// TwinCAT 3 PLC project Theseus
// ProgramVersion: 3.1.4024.0
// libraries:
//   Tc2_ControllerToolbox, * (Beckhoff Automation GmbH)
//   Tc2_MC2, * (Beckhoff Automation GmbH)
//   Tc2_ModbusRTU, * (Beckhoff Automation GmbH)
//   Tc2_Standard, * (Beckhoff Automation GmbH)
//   Tc2_System, * (Beckhoff Automation GmbH)
//   Tc2_Utilities, * (Beckhoff Automation GmbH)
//   Tc3_Module, * (Beckhoff Automation GmbH)
//   Tc2_OpcUa,3.3.2.0,Beckhoff Automation GmbH
// project tree:
//   Data_Types/ E_MachineState.TcDUT, E_PIDMode.TcDUT (not stored), E_LMH.TcDUT, E_ProductType.TcDUT, E_Status.TcDUT
//   GVLs/ Global_Alarms.TcGVL, Global_Constants.TcGVL, P0_Global_Variables.TcGVL
//   / PlcTask.TcTTO (not stored)
//   POUs/ FB_Reactor.TcPOU, FB_Reactor_Set.TcPOU, MAIN.TcPOU, P_Alarms.TcPOU, P_M01.TcPOU, P_U01.TcPOU
//   POUs/Functions/ F_AnalogIn.TcPOU (not stored), F_Concat3.TcPOU (not stored), F_Concat4.TcPOU, F_HighestInt.TcPOU (not stored), F_IEConvert.TcPOU, F_LowestReal.TcPOU (not stored), F_HighestReal.TcPOU, F_LowMidHigh.TcPOU, F_Temperature.TcPOU (not stored), F_SetProcess.TcPOU (not stored), F_ValveClear.TcPOU
//   POUs/Function_Blocks/ FB_Analog_Out.TcPOU, FB_ChangeOfValue.TcPOU, FB_Door_Closed.TcPOU, FB_Integer_Out.TcPOU, FB_MovingAverage.TcPOU, FB_PI_Control.TcPOU, FB_RateOfChange.TcPOU, FB_Temperature.TcPOU, FB_ValveError.TcPOU, FB_VFD.TcPOU
// real-time tasks:
//   TASK PlcTask: cycle T#10ms, priority 20, ADS port 350
// I/O:
//   DEVICE Device 2 (EtherCAT) (disabled), AmsNetId 192.168.1.143.3.1
//     Term 1 (EK1100) [EK1100 EtherCAT Coupler (2A E-Bus)]
//       Term 2 (EL6070) [EL6070 1Ch. Licensing-Terminal]
//       Term 3 (EL1008) [EL1008 8Ch. Dig. Input 24V, 3ms]
//       Term 4 (EL1008) [EL1008 8Ch. Dig. Input 24V, 3ms]
//       Term 5 (EL1008) [EL1008 8Ch. Dig. Input 24V, 3ms]
//       Term 6 (EL1008) [EL1008 8Ch. Dig. Input 24V, 3ms]
//       Term 7 (EL1008) [EL1008 8Ch. Dig. Input 24V, 3ms]
//       Term 8 (EL1008) [EL1008 8Ch. Dig. Input 24V, 3ms]
//       Term 9 (EL1008) [EL1008 8Ch. Dig. Input 24V, 3ms]
//       Term 10 (EL2008) [EL2008 8Ch. Dig. Output 24V, 0.5A]
//       Term 11 (EL2008) [EL2008 8Ch. Dig. Output 24V, 0.5A]
//       Term 12 (EL2008) [EL2008 8Ch. Dig. Output 24V, 0.5A]
//       Term 13 (EL2008) [EL2008 8Ch. Dig. Output 24V, 0.5A]
//       Term 14 (EL2008) [EL2008 8Ch. Dig. Output 24V, 0.5A]
//       Term 15 (EL2008) [EL2008 8Ch. Dig. Output 24V, 0.5A]
//       Term 16 (EL2008) [EL2008 8Ch. Dig. Output 24V, 0.5A]
//       Term 18 (EL9410) [EL9410 E-Bus Power Supplier  (Diagnostics)]
//       Term 19 (EL3058) [EL3058 8Ch. Ana. Input 4-20mA]
//       Term 20 (EL3058) [EL3058 8Ch. Ana. Input 4-20mA]
//       Term 21 (EL3058) [EL3058 8Ch. Ana. Input 4-20mA]
//       Term 22 (EL3058) [EL3058 8Ch. Ana. Input 4-20mA]
//       Term 23 (EL3058) [EL3058 8Ch. Ana. Input 4-20mA]
//       Term 24 (EL4122) [EL4122 2Ch. Ana. Output  4-20mA, 16bit]
//       Term 25 (EL3318) [EL3318 8Ch. Ana Input Thermocouple (TC)]
//       Term 26 (EL3318) [EL3318 8Ch. Ana Input Thermocouple (TC)]
//       Term 27 (EL3318) [EL3318 8Ch. Ana Input Thermocouple (TC)]
//       Term 28 (EL3318) [EL3318 8Ch. Ana Input Thermocouple (TC)]
//       Term 29 (EL3318) [EL3318 8Ch. Ana Input Thermocouple (TC)]
//       Term 30 (EL9410) [EL9410 E-Bus Power Supplier  (Diagnostics)]
//       Term 31 (EL3214) [EL3214 4Ch. Ana. Input PT100 (RTD)]
//       Term 32 (EK1110) [EK1110 EtherCAT extension]
//     Term 33 (EK1100) [EK1100 EtherCAT Coupler (2A E-Bus)]
//       Term 34 (EL3058) [EL3058 8Ch. Ana. Input 4-20mA]
//       Term 35 (EL3058) [EL3058 8Ch. Ana. Input 4-20mA]
//       Term 36 (EL2008) [EL2008 8Ch. Dig. Output 24V, 0.5A]
//       Term 37 (EL2008) [EL2008 8Ch. Dig. Output 24V, 0.5A]
//       Term 38 (EK1122) [EK1122 2 port EtherCAT junction]
//         Box 40 (Commander C200 Open Loop) [Commander C200 Open Loop]
//       Term 39 (EL9011) [EL9011 End Terminal]
// variable links:
//   Theseus/Theseus Instance <-> Device 2 (EtherCAT)/Term 1 (EK1100)/Term 10 (EL2008)
//     PlcTask Outputs/P_M01.rs1.r1.AT_01_pump <-> Channel 3/Output
//     PlcTask Outputs/P_M01.rs1.r1.AT_03_pump <-> Channel 1/Output
//     PlcTask Outputs/P_M01.rs1.r1.AT_01_sol <-> Channel 4/Output
//     PlcTask Outputs/P_M01.rs1.r1.AT_03_sol <-> Channel 2/Output
//     PlcTask Outputs/P_M01.rs1.r1.XV_02 <-> Channel 5/Output
//     PlcTask Outputs/P_M01.rs1.r1.XV_09 <-> Channel 6/Output
//     PlcTask Outputs/P_M01.rs1.r1.outlet_door_far_clamps_extend_valve <-> Channel 7/Output
//     PlcTask Outputs/P_M01.rs1.r1.outlet_door_far_clamps_retract_valve <-> Channel 8/Output
//   Theseus/Theseus Instance <-> Device 2 (EtherCAT)/Term 1 (EK1100)/Term 11 (EL2008)
//     PlcTask Outputs/P_M01.rs1.r1.inlet_door_far_clamps_extend_valve <-> Channel 3/Output
//     PlcTask Outputs/P_M01.rs1.r1.inlet_door_far_clamps_retract_valve <-> Channel 4/Output
//     PlcTask Outputs/P_M01.rs1.r1.inlet_door_near_clamps_extend_valve <-> Channel 5/Output
//     PlcTask Outputs/P_M01.rs1.r1.inlet_door_near_clamps_retract_valve <-> Channel 6/Output
//     PlcTask Outputs/P_M01.rs1.r1.outlet_door_close_valve <-> Channel 8/Output
//     PlcTask Outputs/P_M01.rs1.r1.outlet_door_near_clamps_extend_valve <-> Channel 1/Output
//     PlcTask Outputs/P_M01.rs1.r1.outlet_door_near_clamps_retract_valve <-> Channel 2/Output
//     PlcTask Outputs/P_M01.rs1.r1.outlet_door_open_valve <-> Channel 7/Output
//   Theseus/Theseus Instance <-> Device 2 (EtherCAT)/Term 1 (EK1100)/Term 12 (EL2008)
//     PlcTask Outputs/P_M01.rs1.XV_04 <-> Channel 3/Output
//     PlcTask Outputs/P_M01.rs1.XV_05 <-> Channel 4/Output
//     PlcTask Outputs/P_M01.rs1.XV_06 <-> Channel 5/Output
//     PlcTask Outputs/P_M01.rs1.XV_07 <-> Channel 6/Output
//     PlcTask Outputs/P_M01.rs1.XV_08 <-> Channel 7/Output
//     PlcTask Outputs/P_M01.rs1.r1.inlet_door_close_valve <-> Channel 2/Output
//     PlcTask Outputs/P_M01.rs1.r1.inlet_door_open_valve <-> Channel 1/Output
//   Theseus/Theseus Instance <-> Device 2 (EtherCAT)/Term 1 (EK1100)/Term 13 (EL2008)
//     PlcTask Outputs/P_U01.XV_03 <-> Channel 4/Output
//     PlcTask Outputs/P_U01.XV_04 <-> Channel 3/Output
//     PlcTask Outputs/P_U01.XV_06 <-> Channel 1/Output
//     PlcTask Outputs/P_U01.XV_12 <-> Channel 6/Output
//   Theseus/Theseus Instance <-> Device 2 (EtherCAT)/Term 1 (EK1100)/Term 14 (EL2008)
//     PlcTask Outputs/P_U01.XV_10 <-> Channel 1/Output
//     PlcTask Outputs/P_U01.XV_11 <-> Channel 4/Output
//     PlcTask Outputs/P_U01.XV_13 <-> Channel 2/Output
//     PlcTask Outputs/P_U01.XV_14 <-> Channel 5/Output
//   Theseus/Theseus Instance <-> Device 2 (EtherCAT)/Term 1 (EK1100)/Term 19 (EL3058)
//     PlcTask Inputs/P_M01.rs1.r1.AT_01 <-> AI Standard Channel 3/Value
//     PlcTask Inputs/P_M01.rs1.r1.AT_02 <-> AI Standard Channel 2/Value
//     PlcTask Inputs/P_M01.rs1.r1.AT_03 <-> AI Standard Channel 1/Value
//     PlcTask Inputs/P_M01.rs1.r1.AT_04 <-> AI Standard Channel 4/Value
//     PlcTask Inputs/P_M01.rs1.r1.AT_01_error <-> AI Standard Channel 1/Status/Error
//     PlcTask Inputs/P_M01.rs1.r1.AT_02_error <-> AI Standard Channel 2/Status/Error
//     PlcTask Inputs/P_M01.rs1.r1.AT_03_error <-> AI Standard Channel 3/Status/Error
//     PlcTask Inputs/P_M01.rs1.r1.AT_04_error <-> AI Standard Channel 4/Status/Error
//     PlcTask Inputs/P_M01.rs1.r1.FT_01 <-> AI Standard Channel 5/Value
//     PlcTask Inputs/P_M01.rs1.r1.FT_01_error <-> AI Standard Channel 5/Status/Error
//     PlcTask Inputs/P_M01.rs1.r1.PDT_01 <-> AI Standard Channel 6/Value
//     PlcTask Inputs/P_M01.rs1.r1.PDT_02 <-> AI Standard Channel 7/Value
//     PlcTask Inputs/P_M01.rs1.r1.PDT_03 <-> AI Standard Channel 8/Value
//     PlcTask Inputs/P_M01.rs1.r1.PDT_01_error <-> AI Standard Channel 6/Status/Error
//     PlcTask Inputs/P_M01.rs1.r1.PDT_02_error <-> AI Standard Channel 7/Status/Error
//     PlcTask Inputs/P_M01.rs1.r1.PDT_03_error <-> AI Standard Channel 8/Status/Error
//   Theseus/Theseus Instance <-> Device 2 (EtherCAT)/Term 1 (EK1100)/Term 20 (EL3058)
//     PlcTask Inputs/P_M01.rs1.FT_02 <-> AI Standard Channel 2/Value
//     PlcTask Inputs/P_M01.rs1.FT_02_error <-> AI Standard Channel 2/Status/Error
//     PlcTask Inputs/P_M01.rs1.PT_02 <-> AI Standard Channel 3/Value
//     PlcTask Inputs/P_M01.rs1.PT_02_error <-> AI Standard Channel 3/Status/Error
//     PlcTask Inputs/P_M01.rs1.r1.PT_01 <-> AI Standard Channel 1/Value
//     PlcTask Inputs/P_M01.rs1.r1.PT_01_error <-> AI Standard Channel 1/Status/Error
//     PlcTask Inputs/P_U01.WI_01 <-> AI Standard Channel 4/Value
//     PlcTask Inputs/P_U01.WI_02 <-> AI Standard Channel 5/Value
//     PlcTask Inputs/P_U01.WI_03 <-> AI Standard Channel 6/Value
//     PlcTask Inputs/P_U01.WI_01_error <-> AI Standard Channel 4/Status/Error
//     PlcTask Inputs/P_U01.WI_02_error <-> AI Standard Channel 5/Status/Error
//     PlcTask Inputs/P_U01.WI_03_error <-> AI Standard Channel 6/Status/Error
//   Theseus/Theseus Instance <-> Device 2 (EtherCAT)/Term 1 (EK1100)/Term 21 (EL3058)
//     PlcTask Inputs/P_U01.AT_02 <-> AI Standard Channel 6/Value
//     PlcTask Inputs/P_U01.AT_03 <-> AI Standard Channel 7/Value
//     PlcTask Inputs/P_U01.AT_02_error <-> AI Standard Channel 6/Status/Error
//     PlcTask Inputs/P_U01.AT_03_error <-> AI Standard Channel 7/Status/Error
//     PlcTask Inputs/P_U01.FT_02 <-> AI Standard Channel 8/Value
//     PlcTask Inputs/P_U01.FT_04 <-> AI Standard Channel 1/Value
//     PlcTask Inputs/P_U01.FT_07 <-> AI Standard Channel 5/Value
//     PlcTask Inputs/P_U01.FT_02_error <-> AI Standard Channel 8/Status/Error
//     PlcTask Inputs/P_U01.FT_04_error <-> AI Standard Channel 1/Status/Error
//     PlcTask Inputs/P_U01.FT_07_error <-> AI Standard Channel 5/Status/Error
//     PlcTask Inputs/P_U01.LT_02 <-> AI Standard Channel 4/Value
//     PlcTask Inputs/P_U01.LT_02_error <-> AI Standard Channel 4/Status/Error
//     PlcTask Inputs/P_U01.PCV_01_position <-> AI Standard Channel 3/Value
//     PlcTask Inputs/P_U01.PT_04 <-> AI Standard Channel 2/Value
//     PlcTask Inputs/P_U01.PT_04_error <-> AI Standard Channel 2/Status/Error
//     PlcTask Inputs/P_U01.vacuum_pres_control_valve_position_error <-> AI Standard Channel 3/Status/Error
//   Theseus/Theseus Instance <-> Device 2 (EtherCAT)/Term 1 (EK1100)/Term 22 (EL3058)
//     PlcTask Inputs/P_U01.FT_05 <-> AI Standard Channel 1/Value
//     PlcTask Inputs/P_U01.FT_06 <-> AI Standard Channel 4/Value
//     PlcTask Inputs/P_U01.FT_08 <-> AI Standard Channel 7/Value
//     PlcTask Inputs/P_U01.FT_05_error <-> AI Standard Channel 1/Status/Error
//     PlcTask Inputs/P_U01.FT_06_error <-> AI Standard Channel 4/Status/Error
//     PlcTask Inputs/P_U01.FT_08_error <-> AI Standard Channel 7/Status/Error
//     PlcTask Inputs/P_U01.LT_01 <-> AI Standard Channel 2/Value
//     PlcTask Inputs/P_U01.LT_01_error <-> AI Standard Channel 2/Status/Error
//     PlcTask Inputs/P_U01.PCV_02_position <-> AI Standard Channel 3/Value
//     PlcTask Inputs/P_U01.PDT_04 <-> AI Standard Channel 6/Value
//     PlcTask Inputs/P_U01.PDT_04_error <-> AI Standard Channel 6/Status/Error
//     PlcTask Inputs/P_U01.PT_07 <-> AI Standard Channel 5/Value
//     PlcTask Inputs/P_U01.PT_07_error <-> AI Standard Channel 5/Status/Error
//   Theseus/Theseus Instance <-> Device 2 (EtherCAT)/Term 1 (EK1100)/Term 24 (EL4122)
//     PlcTask Outputs/P_U01.PCV_01 <-> Channel 1/Output
//     PlcTask Outputs/P_U01.PCV_02 <-> Channel 2/Output
//   Theseus/Theseus Instance <-> Device 2 (EtherCAT)/Term 1 (EK1100)/Term 25 (EL3318)
//     PlcTask Inputs/P_M01.rs1.r1._01_TT_01 <-> TC Channel 1/Value
//     PlcTask Inputs/P_M01.rs1.r1._01_TT_03 <-> TC Channel 2/Value
//     PlcTask Inputs/P_M01.rs1.r1._02_TT_01 <-> TC Channel 3/Value
//     PlcTask Inputs/P_M01.rs1.r1._02_TT_03 <-> TC Channel 4/Value
//     PlcTask Inputs/P_M01.rs1.r1._03_TT_01 <-> TC Channel 5/Value
//     PlcTask Inputs/P_M01.rs1.r1._03_TT_03 <-> TC Channel 6/Value
//     PlcTask Inputs/P_M01.rs1.r1._04_TT_01 <-> TC Channel 7/Value
//     PlcTask Inputs/P_M01.rs1.r1._04_TT_03 <-> TC Channel 8/Value
//     PlcTask Inputs/P_M01.rs1.r1._01_TT_01_Error <-> TC Channel 1/Status/Error
//     PlcTask Inputs/P_M01.rs1.r1._01_TT_03_Error <-> TC Channel 2/Status/Error
//     PlcTask Inputs/P_M01.rs1.r1._02_TT_01_Error <-> TC Channel 3/Status/Error
//     PlcTask Inputs/P_M01.rs1.r1._02_TT_03_Error <-> TC Channel 4/Status/Error
//     PlcTask Inputs/P_M01.rs1.r1._03_TT_01_Error <-> TC Channel 5/Status/Error
//     PlcTask Inputs/P_M01.rs1.r1._03_TT_03_Error <-> TC Channel 6/Status/Error
//     PlcTask Inputs/P_M01.rs1.r1._04_TT_01_Error <-> TC Channel 7/Status/Error
//     PlcTask Inputs/P_M01.rs1.r1._04_TT_03_Error <-> TC Channel 8/Status/Error
//   Theseus/Theseus Instance <-> Device 2 (EtherCAT)/Term 1 (EK1100)/Term 26 (EL3318)
//     PlcTask Inputs/P_M01.rs1.r1._05_TT_01 <-> TC Channel 1/Value
//     PlcTask Inputs/P_M01.rs1.r1._05_TT_03 <-> TC Channel 2/Value
//     PlcTask Inputs/P_M01.rs1.r1._06_TT_01 <-> TC Channel 3/Value
//     PlcTask Inputs/P_M01.rs1.r1._06_TT_03 <-> TC Channel 4/Value
//     PlcTask Inputs/P_M01.rs1.r1._07_TT_01 <-> TC Channel 5/Value
//     PlcTask Inputs/P_M01.rs1.r1._07_TT_03 <-> TC Channel 6/Value
//     PlcTask Inputs/P_M01.rs1.r1._08_TT_01 <-> TC Channel 7/Value
//     PlcTask Inputs/P_M01.rs1.r1._08_TT_03 <-> TC Channel 8/Value
//     PlcTask Inputs/P_M01.rs1.r1._05_TT_01_Error <-> TC Channel 1/Status/Error
//     PlcTask Inputs/P_M01.rs1.r1._05_TT_03_Error <-> TC Channel 2/Status/Error
//     PlcTask Inputs/P_M01.rs1.r1._06_TT_01_Error <-> TC Channel 3/Status/Error
//     PlcTask Inputs/P_M01.rs1.r1._06_TT_03_Error <-> TC Channel 4/Status/Error
//     PlcTask Inputs/P_M01.rs1.r1._07_TT_01_Error <-> TC Channel 5/Status/Error
//     PlcTask Inputs/P_M01.rs1.r1._07_TT_03_Error <-> TC Channel 6/Status/Error
//     PlcTask Inputs/P_M01.rs1.r1._08_TT_01_Error <-> TC Channel 7/Status/Error
//     PlcTask Inputs/P_M01.rs1.r1._08_TT_03_Error <-> TC Channel 8/Status/Error
//   Theseus/Theseus Instance <-> Device 2 (EtherCAT)/Term 1 (EK1100)/Term 27 (EL3318)
//     PlcTask Inputs/P_M01.rs1.r1._09_TT_01 <-> TC Channel 1/Value
//     PlcTask Inputs/P_M01.rs1.r1._09_TT_03 <-> TC Channel 2/Value
//     PlcTask Inputs/P_M01.rs1.r1._10_TT_01 <-> TC Channel 3/Value
//     PlcTask Inputs/P_M01.rs1.r1._10_TT_03 <-> TC Channel 4/Value
//     PlcTask Inputs/P_M01.rs1.r1._11_TT_01 <-> TC Channel 5/Value
//     PlcTask Inputs/P_M01.rs1.r1._11_TT_03 <-> TC Channel 6/Value
//     PlcTask Inputs/P_M01.rs1.r1._12_TT_01 <-> TC Channel 7/Value
//     PlcTask Inputs/P_M01.rs1.r1._12_TT_03 <-> TC Channel 8/Value
//     PlcTask Inputs/P_M01.rs1.r1._09_TT_01_Error <-> TC Channel 1/Status/Error
//     PlcTask Inputs/P_M01.rs1.r1._09_TT_03_Error <-> TC Channel 2/Status/Error
//     PlcTask Inputs/P_M01.rs1.r1._10_TT_01_Error <-> TC Channel 3/Status/Error
//     PlcTask Inputs/P_M01.rs1.r1._10_TT_03_Error <-> TC Channel 4/Status/Error
//     PlcTask Inputs/P_M01.rs1.r1._11_TT_01_Error <-> TC Channel 5/Status/Error
//     PlcTask Inputs/P_M01.rs1.r1._11_TT_03_Error <-> TC Channel 6/Status/Error
//     PlcTask Inputs/P_M01.rs1.r1._12_TT_01_Error <-> TC Channel 7/Status/Error
//     PlcTask Inputs/P_M01.rs1.r1._12_TT_03_Error <-> TC Channel 8/Status/Error
//   Theseus/Theseus Instance <-> Device 2 (EtherCAT)/Term 1 (EK1100)/Term 29 (EL3318)
//     PlcTask Inputs/P_M01.rs1.TT_01 <-> TC Channel 1/Value
//     PlcTask Inputs/P_M01.rs1.TT_01_error <-> TC Channel 1/Status/Error
//     PlcTask Inputs/P_U01.TT_03 <-> TC Channel 2/Value
//     PlcTask Inputs/P_U01.TT_06 <-> TC Channel 5/Value
//     PlcTask Inputs/P_U01.TT_10 <-> TC Channel 3/Value
//     PlcTask Inputs/P_U01.TT_11 <-> TC Channel 4/Value
//     PlcTask Inputs/P_U01.TT_03_error <-> TC Channel 2/Status/Error
//     PlcTask Inputs/P_U01.TT_06_error <-> TC Channel 5/Status/Error
//     PlcTask Inputs/P_U01.TT_10_error <-> TC Channel 3/Status/Error
//     PlcTask Inputs/P_U01.TT_11_error <-> TC Channel 4/Status/Error
//   Theseus/Theseus Instance <-> Device 2 (EtherCAT)/Term 1 (EK1100)/Term 3 (EL1008)
//     PlcTask Inputs/P_M01.rs1.r1.outlet_door_far_clamps_extended <-> Channel 6/Input
//     PlcTask Inputs/P_M01.rs1.r1.outlet_door_far_closed_ls <-> Channel 4/Input
//     PlcTask Inputs/P_M01.rs1.r1.outlet_door_far_open_ls <-> Channel 3/Input
//     PlcTask Inputs/P_M01.rs1.r1.outlet_door_near_clamps_extended <-> Channel 5/Input
//     PlcTask Inputs/P_M01.rs1.r1.outlet_door_near_closed_ls <-> Channel 2/Input
//     PlcTask Inputs/P_M01.rs1.r1.outlet_door_near_open_ls <-> Channel 1/Input
//     PlcTask Inputs/P_M01.rs1.r1.repres_valve_closed <-> Channel 8/Input
//     PlcTask Inputs/P_M01.rs1.r1.repres_valve_open <-> Channel 7/Input
//   Theseus/Theseus Instance <-> Device 2 (EtherCAT)/Term 1 (EK1100)/Term 31 (EL3214)
//     PlcTask Inputs/P_M01.rs1.r1.TT_04 <-> RTD Inputs Channel 2/Value
//     PlcTask Inputs/P_M01.rs1.r1.TT_05 <-> RTD Inputs Channel 1/Value
//     PlcTask Inputs/P_M01.rs1.r1.TT_04_error <-> RTD Inputs Channel 2/Status/Error
//     PlcTask Inputs/P_M01.rs1.r1.TT_05_error <-> RTD Inputs Channel 1/Status/Error
//     PlcTask Inputs/P_U01.TT_02 <-> RTD Inputs Channel 3/Value
//     PlcTask Inputs/P_U01.TT_02_error <-> RTD Inputs Channel 3/Status/Error
//   Theseus/Theseus Instance <-> Device 2 (EtherCAT)/Term 1 (EK1100)/Term 4 (EL1008)
//     PlcTask Inputs/P_M01.rs1.r1.inlet_door_far_clamps_extended <-> Channel 6/Input
//     PlcTask Inputs/P_M01.rs1.r1.inlet_door_far_closed_ls <-> Channel 4/Input
//     PlcTask Inputs/P_M01.rs1.r1.inlet_door_far_open_ls <-> Channel 3/Input
//     PlcTask Inputs/P_M01.rs1.r1.inlet_door_near_clamps_extended <-> Channel 5/Input
//     PlcTask Inputs/P_M01.rs1.r1.inlet_door_near_closed_ls <-> Channel 2/Input
//     PlcTask Inputs/P_M01.rs1.r1.inlet_door_near_open_ls <-> Channel 1/Input
//     PlcTask Inputs/P_M01.rs1.reactor_drain_vessel_lsh <-> Channel 8/Input
//     PlcTask Inputs/P_M01.rs1.reactor_drain_vessel_lsl <-> Channel 7/Input
//   Theseus/Theseus Instance <-> Device 2 (EtherCAT)/Term 1 (EK1100)/Term 5 (EL1008)
//     PlcTask Inputs/P_M01.rs1.condensate_valve_closed <-> Channel 6/Input
//     PlcTask Inputs/P_M01.rs1.condensate_valve_open <-> Channel 5/Input
//     PlcTask Inputs/P_M01.rs1.dead_air_valve_closed <-> Channel 2/Input
//     PlcTask Inputs/P_M01.rs1.dead_air_valve_open <-> Channel 1/Input
//     PlcTask Inputs/P_M01.rs1.product_iso_valve_closed <-> Channel 4/Input
//     PlcTask Inputs/P_M01.rs1.product_iso_valve_open <-> Channel 3/Input
//     PlcTask Inputs/P_M01.rs1.steam_iso_valve_closed <-> Channel 8/Input
//     PlcTask Inputs/P_M01.rs1.steam_iso_valve_open <-> Channel 7/Input
//   Theseus/Theseus Instance <-> Device 2 (EtherCAT)/Term 1 (EK1100)/Term 6 (EL1008)
//     PlcTask Inputs/P_M01.rs1.steam_bypass_valve_closed <-> Channel 2/Input
//     PlcTask Inputs/P_M01.rs1.steam_bypass_valve_open <-> Channel 1/Input
//   Theseus/Theseus Instance <-> Device 2 (EtherCAT)/Term 1 (EK1100)/Term 7 (EL1008)
//     PlcTask Inputs/P_U01.knockout_drain_valve_closed <-> Channel 4/Input
//     PlcTask Inputs/P_U01.knockout_drain_valve_open <-> Channel 3/Input
//     PlcTask Inputs/P_U01.product_condensate_drum_lsh <-> Channel 2/Input
//     PlcTask Inputs/P_U01.product_condensate_drum_lsl <-> Channel 1/Input
//     PlcTask Inputs/P_U01.vacuum_pump_bypass_valve_closed <-> Channel 6/Input
//     PlcTask Inputs/P_U01.vacuum_pump_bypass_valve_open <-> Channel 5/Input
//     PlcTask Inputs/P_U01.vacuum_pump_inlet_valve_closed <-> Channel 8/Input
//     PlcTask Inputs/P_U01.vacuum_pump_inlet_valve_open <-> Channel 7/Input
//   Theseus/Theseus Instance <-> Device 2 (EtherCAT)/Term 1 (EK1100)/Term 8 (EL1008)
//     PlcTask Inputs/P_U01.dead_air_inlet_valve_closed <-> Channel 2/Input
//     PlcTask Inputs/P_U01.dead_air_inlet_valve_open <-> Channel 1/Input
//     PlcTask Inputs/P_U01.product_line_ambient_valve_ambient <-> Channel 5/Input
//     PlcTask Inputs/P_U01.product_line_ambient_valve_product <-> Channel 6/Input
//     PlcTask Inputs/P_U01.separator_drain_valve_closed <-> Channel 4/Input
//     PlcTask Inputs/P_U01.separator_drain_valve_open <-> Channel 3/Input
//   Theseus/Theseus Instance <-> Device 2 (EtherCAT)/Term 33 (EK1100)/Term 34 (EL3058)
//     PlcTask Inputs/P_U01.IT1 <-> AI Standard Channel 5/Value
//     PlcTask Inputs/P_U01.IT2 <-> AI Standard Channel 6/Value
//     PlcTask Inputs/P_U01.IT3 <-> AI Standard Channel 7/Value
//     PlcTask Inputs/P_U01.IT4 <-> AI Standard Channel 8/Value
//     PlcTask Inputs/P_U01.VT1 <-> AI Standard Channel 1/Value
//     PlcTask Inputs/P_U01.VT2 <-> AI Standard Channel 2/Value
//     PlcTask Inputs/P_U01.VT3 <-> AI Standard Channel 3/Value
//     PlcTask Inputs/P_U01.VT4 <-> AI Standard Channel 4/Value
//     PlcTask Inputs/P_U01.l1_current_120_error <-> AI Standard Channel 8/Status/Error
//     PlcTask Inputs/P_U01.l1_current_240_error <-> AI Standard Channel 5/Status/Error
//     PlcTask Inputs/P_U01.l2_current_240_error <-> AI Standard Channel 6/Status/Error
//     PlcTask Inputs/P_U01.l3_current_240_error <-> AI Standard Channel 7/Status/Error
//     PlcTask Inputs/P_U01.l1_voltage_120_error <-> AI Standard Channel 4/Status/Error
//     PlcTask Inputs/P_U01.l1_voltage_240_error <-> AI Standard Channel 1/Status/Error
//     PlcTask Inputs/P_U01.l2_voltage_240_error <-> AI Standard Channel 2/Status/Error
//     PlcTask Inputs/P_U01.l3_voltage_240_error <-> AI Standard Channel 3/Status/Error
//   Theseus/Theseus Instance <-> Device 2 (EtherCAT)/Term 33 (EK1100)/Term 36 (EL2008)
//     PlcTask Outputs/P_U01.B_01 <-> Channel 5/Output
//     PlcTask Outputs/P_U01.P_01 <-> Channel 4/Output
//     PlcTask Outputs/P_U01.P_02 <-> Channel 2/Output
//     PlcTask Outputs/P_U01.P_03 <-> Channel 1/Output
//     PlcTask Outputs/P_U01.P_05 <-> Channel 7/Output
//     PlcTask Outputs/P_U01.P_06 <-> Channel 3/Output
//     PlcTask Outputs/P_U01.X_01 <-> Channel 8/Output
//     PlcTask Outputs/P_U01.boiler_reset <-> Channel 6/Output
//   Theseus/Theseus Instance <-> Device 2 (EtherCAT)/Term 33 (EK1100)/Term 37 (EL2008)
//     PlcTask Outputs/P_U01.E_01 <-> Channel 2/Output
//     PlcTask Outputs/P_U01.P_04 <-> Channel 1/Output
//   Theseus/Theseus Instance <-> Device 2 (EtherCAT)/Term 33 (EK1100)/Term 38 (EK1122)/Box 40 (Commander C200 Open Loop)
//     PlcTask Inputs/P_M01.rs1.r1.fan_vfd_current <-> Transmit PDO Mapping 6/vfd output current param 04_001
//     PlcTask Inputs/P_M01.rs1.r1.fan_vfd_ecat_state <-> WcState/WcState
//     PlcTask Inputs/P_M01.rs1.r1.fan_vfd_status <-> Transmit PDO Mapping 6/Status word
//     PlcTask Inputs/P_M01.rs1.r1.fan_vfd_velocity <-> Transmit PDO Mapping 6/vl velocity actual value
//     PlcTask Outputs/P_M01.rs1.r1.fan_vfd_control <-> Receive PDO Mapping 6/Control word
//     PlcTask Outputs/P_M01.rs1.r1.fan_vfd_target_vel <-> Receive PDO Mapping 6/vl target velocity

// ---- Data_Types/E_MachineState.TcDUT
// Theseus - E_MachineState
// Rev 1.0 - December 2, 2024

TYPE E_MachineState :
(
	eStateOff						:= 0,
	eIdle,
	eDoorCycle,
	ePositivePressure,
	eRepressurization,
	eAdsorption,
	eEvacuation,
	eDesorption,
	eBypass,
	eSingleProcessAuto,
	eChangeState,
	ePause
);
END_TYPE

// ---- Data_Types/E_LMH.TcDUT
// Theseus - E_LMH
// Rev 1.0 - March 14, 2024

TYPE E_LMH :
(
	eLow			 													:= 0,
	eMid,
	eHigh
);
END_TYPE

// ---- Data_Types/E_ProductType.TcDUT
// Theseus - E_ProductType
// Rev 1.0 - June 15, 2024

TYPE E_ProductType :
(
	eAmbient			 												:= 0,
	eProduct
);
END_TYPE

// ---- Data_Types/E_Status.TcDUT
// Theseus - E_Status
// Rev 1.0 - December 2, 2024

TYPE E_Status :
(
	eSystem_Idle						:= 0,
	e1,
	e2,
	eWarmup_Running,			
	eSteamBypass_Running,		
	eDoorCycle_Running,		
	ePositivePressure_Running,	
	eRepressurization_Running,	
	eAdsorption_Running,		
	eEvacuation_Running,		
	eDesorption_Running,
	eBypass_Running,
	eShutting_Down,				
	ePressureTest_Running,		
	e12,                        
	eWarmup_Error,				
	eSteamBypass_Error,			
	eDoor_Cycle_Error,			
	ePositivePressure_Error,	
	eRepressurization_Error,	
	eAdsorption_Error,			
	eEvacuation_Error,			
	eDesorption_Error,
	eShutdown_Error,			
	ePressureTest_Error,		
	e21,                        
	e22,                        
	eWarmup_Complete,			
	eSteamBypass_Complete,		
	eDoorCycle_Complete,         
	ePositivePressure_Complete,	
	eRepressurization_Complete,	
	eAdsorption_Complete,		
	eEvacuation_Complete,		
	eDesorption_Complete,
	eBypass_Complete,		
	eShutdown_Complete,			
	ePressureTest_Complete,		
	e32,                        
	eStopping_Process,			
	eResetting,					
	eSaving_Data				
);
END_TYPE

// ---- GVLs/Global_Alarms.TcGVL
// Theseus - Global_Alarms
// Rev 1.0 - December 3, 2024

VAR_GLOBAL
	
	giAlarmCount														: INT		:= 0;
	gsAlarms															: ARRAY[0.._ALARM_COUNT] OF STRING;
	gsMessages															: ARRAY[0.._ALARM_COUNT] OF STRING;

	gsClampsNotExtendedError											: STRING	:= 'Clamps not extended';
	gsClampsNotRetractedError											: STRING	:= 'Clamps not retracted';
	gsDoorsNotSelectedError												: STRING	:= 'No doors were selected';
	gsGasketNotActivatedError											: STRING	:= 'Gasket not activated';
	gsInletDoorNotClosedError											: STRING	:= 'Inlet door not closed';
	gsInletDoorNotOpenError												: STRING	:= 'Inlet door not open';
	gsOutletDoorNotClosedError											: STRING	:= 'Outlet door not closed';
	gsOutletDoorNotOpenError											: STRING	:= 'Outlet door not open';
	gsPositivePressureError												: STRING	:= 'Reactor failed to reach positive pressure set point';
	gsReactorNotAtAmbientPressure										: STRING	:= 'Reactor not at ambient pressure';
	gsUnacceptableReactorLeakRate										: STRING	:= 'Unacceptable reactor positive pressure leak rate';
	gsRepressurizationValveError										: STRING	:= 'Repressurization valve error (XV02)';	

	
	gsAmbientPressureError												: STRING	:= 'Ambient pressure error';
	gsAdsorptionAcceptableButNotIdealTimeError							: STRING	:= 'Adsorption time to cool acceptable but not ideal';
	gsAdsorptionTimeOutError											: STRING	:= 'Adsorption - sorbent failed to cool';
	gsAdsorptionUnacceptableTimeError									: STRING	:= 'Adsorption time to cool unacceptable';
	gsAdsorptionInletCo2LowError										: STRING	:= 'Adsorption inlet co2 concentration low';
	gsAirFlowSensorError												: STRING	:= 'Air flow sensor error (R1 FT01)';
	gsBoilerError														: STRING	:= 'Boiler error';
	gsInletLineTempSensorError											: STRING	:= 'Inlet line temperature sensor error (TT06)';
	gsClampExtendError													: STRING	:= 'Clamp extend error';
	gsClampRetractError													: STRING	:= 'Clamp retract error';
	gsCondensateFlowSensorError											: STRING	:= 'Condensate flow sensor error (FT-04)';
	gsCondenserKODrainageError											: STRING	:= 'Condensate knockout drainage error';
	gsCondensateLslError												: STRING	:= 'Condensate low limit switch error (LS-01)';
	gsCondenserFlowSensorError											: STRING	:= 'Condenser flow sensor error (FT08)';
	gsCondensateProductDrainError										: STRING	:= 'Module product/cooling line not draining';	
	gsCondensateValveError												: STRING	:= 'Condensate valve error (XV06)';
	gsDeadAirInletValveError											: STRING	:= 'Dead air inlet valve error (XV10)';
	gsDeadAirLinePressureError											: STRING	:= 'Dead air line failed to reach desired pressure';
	gsDeadAirValveError													: STRING	:= 'Dead air valve error (XV04)';
	gsDesiredCycleCountError											: STRING	:= 'Desired cycle count error';
	gsDesorptionHighSteamLineTemp										: STRING	:= 'Desorption - High steam line temperature';
	gsDesorptionPurgeLinePressureError									: STRING	:= 'Desorption - Unable to purge';
	gsDoorClampsExtendedError											: STRING	:= 'Door clamps extended';
	gsDoorsNotClosedError												: STRING	:= 'Door not closed error';
	gsDoorsNotOpenError													: STRING	:= 'Door not open error';
	gsFanDiffPresSensorError											: STRING	:= 'Fan differential pressure sensor error (PDT-03)';
	gsFilterDiffPresSensorError											: STRING	:= 'Filter differential pressure sensor error (PDT-01)';
	gsFlowCalibrationDiffPresSensorError								: STRING	:= 'Flow calibration differential pressure sensor error (PDT04)';
	gsHighTempCountError												: STRING	:= 'High Temp Count Error';
	gsInletAirHighTempCountError										: STRING	:= 'Inlet air high temperature count error';
    gsInletCO2SensorError												: STRING	:= 'Inlet CO2 sensor error (AT-01)';
    gsInletH2OSensorError												: STRING	:= 'Inlet H2O sensor error (AT-02)';
	gsInletDoorClampsExtendedError										: STRING	:= 'Inlet door clamps extended error (XV01)'; 
	gsInletDoorClampsRetractedError										: STRING	:= 'Inlet door clamps retracted error (XV01)'; 
	gsNoReactorSetsSelected												: STRING	:= 'No reactor sets selected';
    gsOutletCO2SensorError												: STRING	:= 'Outlet CO2 sensor error (AT-03)';
    gsOutletH2OSensorError												: STRING	:= 'Outlet H2O sensor error (AT-04)';
	gsOutletDoorClampsExtendedError										: STRING	:= 'Outlet door clamps extended error (XV03)'; 
	gsOutletDoorClampsRetractedError									: STRING	:= 'Outlet door clamps retracted error (XV03)'; 
	gsProductVacuumTempSensorError										: STRING	:= 'Product vacuum temperature sensor error (TT-03)';
	gsProductTempSensorError											: STRING	:= 'Product temperature sensor error (TT-02)';
	gsProductCondensateDrainError										: STRING	:= 'Product condensate not draining';
	gsProductCondensateDrainValveError									: STRING	:= 'Product condensate drain valve error';
	gsProductCondensateDrumLshError										: STRING	:= 'Product condensate drum high limit switch error (LS-02)';
	gsProductCondensateDrumLslError										: STRING	:= 'Product condensate drum low limit switch error (LS-01)';
	gsProductLineAmbientValveError										: STRING	:= 'Product line ambient valve error (XV11)';
	gsProductLinePressureSensorError									: STRING	:= 'Product line pressure sensor error (PT02)';
	gsProductLineTempTooLowError										: string	:= 'Product line temperature too low';
	gsProductOutletH2oSensorError										: STRING	:= 'Product outlet h2o sensor error (AT-02B)';
	gsProductOutletCo2SensorError										: STRING	:= 'Product outlet co2 sensor error (AT-02A)';
	gsProductOutletFlowSensorError										: STRING	:= 'Product outlet flow sensor error (FT02)';
	gsProductVacuumBackfeedValveError									: STRING	:= 'Product vacuum backfeed valve error (PCV-01)';
	gsProductVacuumOutletIsoValveError									: STRING	:= 'Product vacuum outlet isolation valve error (XV-05)';
	gsProductVacuumPumpIsoValveError									: STRING	:= 'Product vacuum pump isolation valve error (XV-03)';
	gsProductVacuumPresSensorError										: STRING	:= 'Product vacuum pressure sensor error (PT-05)';
	gsPurgeProductLinePresLowError										: STRING	:= 'Purge product line pressure low error';
	gsProductIsoValveError												: STRING	:= 'Product isolation valve error (XV05)';
	gsProductLinePresSensorError										: STRING	:= 'Product line pressure sensor error (PT-02)';
	gsProductLineTempSensorError										: STRING	:= 'Product line temperature sensor error (TT-01)';
	gsReactorCondensateFlowSensorError									: STRING	:= 'Reactor condensate flow sensor error (FT02)';
	gsReactorDrainError													: STRING	:= 'Reactor not draining';	
	gsReactorDoorClosingError											: STRING	:= 'Failed to close door valves';									// Complete
	gsReactorDoorOpeningError											: STRING	:= 'Failed to open door valves';									// Complete
	gsReactorsAtAmbientPressure											: STRING	:= 'Reactors at ambient pressure';
	gsReactorPressureAboveAcceptableLevelError							: STRING	:= 'Reactor pressure above acceptable level';
	gsReactorPressureAboveDesiredLevelError								: STRING	:= 'Reactor pressure above desired level';
	gsReactorPressureTooHighError										: STRING	:= 'Reactor pressure too high error';
	gsReactorPressureTooLowError										: STRING	:= 'Reactor pressure too low error';
	gsReactorPresSensorError											: STRING	:= 'Reactor pressure sensor error (PT01)';
	gsReactorSetFailedToPressurizeError									: STRING	:= 'Reactor set failed to pressurize';
	gsReactorValvesNotClosedError										: STRING	:= 'Reactor valves are not closed';
	gsRepressurizationError												: STRING	:= 'Repressurization error';	
	gsSorbentDiffPresSensorError										: STRING	:= 'Sorbent differential pressure sensor error (PDT-02)';
	gsSorbentTemperatureError											: STRING	:= 'Sorbent temperatures above safe temperature';
	gsSteamBypassMinFlowRateError										: STRING	:= 'Steam bypass minimum flow rate error';
	gsSteamControlValveError											: STRING	:= 'Steam control valve error (PCV-01)';
	gsSteamIsoValveError												: STRING	:= 'Steam isolation valve error (XV07)';
	gsSteamFailedToPressurizeReactorError								: STRING	:= 'Steam failed to pressurize reactor to purge pressure';
	gsSteamFlowSensorError												: STRING	:= 'Steam flow sensor error (FT05)';
	gsSteamBypassValveError												: STRING	:= 'Steam bypass valve error (XV08)';
	gsSteamPressureHighError											: STRING	:= 'High steam pressure';
	gsSteamPressureLowError												: STRING	:= 'Low steam pressure';
	gsSteamTemperatureLowError											: STRING	:= 'Low steam temperature';
	gsSteamLinePresSensorError											: STRING	:= 'Steam line pressure sensor error (PT07)';
	gsSteamFlowConrolValveError											: STRING	:= 'Steam flow control valve error (PCV02)';
	gsSteamFlowTooLowError												: STRING	:= 'Steam flow too low error';
	gsSteamWaterTankLevelSensorError									: STRING	:= 'Steam water tank level sensor error (LT01)';
	gsTapWaterFeedFlowSensorError										: STRING	:= 'Tap water feed flow sensor error (FT05)';
	gsUnableToEvacuateLinesError										: STRING	:= 'Unable to evacuate lines in time';
	gsVacuumPressureControlValveError									: STRING	:= 'Vacuum pressure control valve error (PCV01)';
	gsVacuumCoolingLoopFlowError										: STRING	:= 'Vacuum cooling loop flow error';
	gsVacuumCoolingLoopTempError										: STRING	:= 'Vacuum cooling loop temperature error';
	gsVacuumCoolingUnacceptableError									: STRING	:= 'Vacuum cooling temperature reached was unacceptable';
	gsVacuumCoolingAcceptableButNotIdealError							: STRING	:= 'Vacuum cooling temperature reached was acceptable but not ideal';
	gsVacuumLinePressureHighError										: STRING	:= 'Vacuum line pressure high';
	gsVacuumPumpWaterFlowSensorError									: STRING	:= 'Vacuum pump water flow sensor error (FT07)';
	gsVacuumPumpWaterTemp1SensorError									: STRING	:= 'Vacuum pump water temperature 1 sensor error (TT10)';
	gsVacuumPressureUnacceptableError									: STRING	:= 'Vacuum pressure reached was unacceptable';
	gsVacuumPressureAcceptableBotNotIdealError							: STRING	:= 'Vacuum pressure reached was acceptable but not ideal';
	gsVacuumPumpBypassValveError										: STRING	:= 'Vacuum pump bypass valve error (XV04)';
	gsVacuumPumpInletValveError											: STRING	:= 'Vacuum pump inlet valve error (XV03)';
	gsVacuumSeparatorLevelSensorError									: STRING	:= 'Vacuum separator level sensor error (LT02)';
	gsVacuumSeparatorDrainError											: STRING	:= 'Vacuum separator drain error';
	gsVacuumSeparatorFillError											: STRING	:= 'Vacuum separator fill error';
	gsWarmupNotRunError													: STRING	:= 'Warmup has not run';
	gsWeatherHumiditySensorError										: STRING	:= 'Weather humidity sensor error (AT-07)';
	gsWeatherPresureSensorError											: STRING	:= 'Weather pressure sensor error (PT-09)';
	gsWaterScale1SensorError											: STRING	:= 'Water Scale 1 sensor error (WI-01)';
	gsWaterScale2SensorError											: STRING	:= 'Water Scale 2 sensor error (WI-02)';
	gsWaterScale3SensorError											: STRING	:= 'Water Scale 3 sensor error (WI-03)';
	
	gsMessageTBD			: STRING	:= 'TBD';
	gsAdsorptionCo2LowCheck												: STRING	:= 'Check inlet co2 sensor';
	gsCheckOperation													: STRING	:= 'Check sensor operation';
	gsExtraRepressurizationTimeAllowed									: STRING	:= 'Extra repressurization time allowed';
	gsPressureDropTestCannotRun											: STRING	:= 'Pressure drop test cannot run';
	gsProcessCannotContinue												: STRING	:= 'Process cannot continue';
	gsProcessCannotRun													: STRING	:= 'Process cannot run';
	gsProcessCannotRunAdsorptionWillContinue							: STRING	:= 'Process cannot run - Adsorption will continue';
	gsProcessStopsAtEOA													: STRING	:= 'Process will stop at end of Adsorption';
	gsProcessStopsAtEOC													: STRING	:= 'Process will stop at end of current cycle';
	gsProcessWillContinue												: STRING	:= 'Process will continue';
	gsProcessComplete													: STRING	:= 'Process complete';
	gsProcessRestart													: STRING	:= 'Process will attempt to restart on next cycle';
	gsReactorIsUnderVacuum												: STRING	:= 'Reactor is under vacuum';
	gsReactorSetCannotRun												: STRING	:= 'Reactor set cannot run';
	gsReactorSetWillContinue											: STRING	:= 'Reactor set will continue';
	gsReactorSetWillPause												: STRING	:= 'Reactor set will pause';
	gsReactorSetWillStop												: STRING	:= 'Reactor set will stop';
	gsReactorSetWillStopAtEndOfCycle									: STRING	:= 'Reactor set will stop at end of cycle';
	gsReactorSetsInEvacuationWillContinue								: STRING	:= 'Reactor sets in Evacuation will finish, others will stop';
	gsReactorSetWillStopEvacWillFinishOthersWillCompleteCycle			: STRING	:= 'Reactor set will stop, Evacuation will finish, others will complete cycle';
	gsRunWarmup															: STRING	:= 'Run warm up';													
	gsSorbentDamaged													: STRING	:= 'Sorbent damaged';
	gsSteamBypassWillContinueWOAdsorption								: STRING	:= 'Steam Bypass will continue without Adsorption';
	gsSystemCannotRun													: STRING	:= 'System cannot run';
	gsSystemWillStop													: STRING	:= 'System will stop';
	gsSystemWillStopAfterDesorption										: STRING	:= 'System will stop after Desorption';
	gsUnableToCloseDoors												: STRING	:= 'Unable to close doors';
	gsUnableToEvacuateReactorSet										: STRING	:= 'Unable to evacuate reactor set';
	gsUserProcessRestart												: STRING	:= 'User must restart for process to continue';
	gsWarmupWillContinue												: STRING	:= 'Warm up will continue';													
	gsWarmupWillContinueWOAdsorption									: STRING	:= 'Warm up will continue without Adsorption';
	gsWarning															: STRING	:= 'Waring - Procees could be affected';

END_VAR

// ---- GVLs/Global_Constants.TcGVL
// Theseus - Global_Constants
// Rev 1.0 - November 4, 2024

VAR_GLOBAL CONSTANT
	
	_DOOR_ACTUATION_TIMEOUT												: REAL		:= 120000;
	_CLAMP_ACTUATION_TIMEOUT											: REAL		:= 10000;
	_VALVE_TIME															: REAL		:= 5000;
	
	_ALARM_COUNT														: INT		:= 100;
	_DRAIN_TIME															: TIME		:= T#3S;
	_DOOR_LATCH_CLOSE_TIME												: TIME		:= T#2S;
	_FAN_SPEED_MAX														: REAL		:= 1765;		// Maximum Fan RPM
	_FAN_SPEED_MIN														: REAL		:= 300;			// Minimum Fan RPM
	_PUMP_SPEED_MAX														: REAL		:= 3540;		// Maximum Pump RPM
	_PUMP_SPEED_MIN														: REAL		:= 200;			// Minimum Pump RPM
	_FAN_DELAY_TIME														: INT		:= 2000;
	_FAN_RS_DELAY_TIME													: INT		:= 15000;
	_PROCESS_COMPLETE_TIME												: REAL		:= 2000;
	_PAUSE_TIME															: REAL		:= 2000;
	_FAN_SHUTDOWN_TIME													: REAL		:= 10000;
	_VALVE_INCREMENT_TIME												: REAL		:= 250;			// Time period for incremental change in valve position (mSecs)
	_STOPPING_TIME														: REAL		:= 2000;
	_VALVE_CLOSED														: INT		:= 3;
	_VALVE_OPEN															: INT		:= 95;
	
	_CURRENT_120_FACTOR													: REAL		:= 655.34;		// =  32767 counts / 50 amps
	_CURRENT_240_FACTOR													: REAL		:= 218.44;      // = 32767 counts / 150 amps
	_CURRENT_BOILER_FACTOR												: REAL 		:= 40.95 * 2 ;	//  = 32767 / 800 Amps * 2 (double coiled)
	_CURRENT_MODULE_FACTOR												: REAL		:= 81.91;		// 0- 800 amps	
	_PERCENT_FACTOR														: REAL		:= 327.67;		// Factor to convert input to output percentage
	_FAN_RPM_FACTOR														: REAL		:= 17.65;		// Factor to convert fan percent input to rpm output (max rpm / 100)
	_PUMP_RPM_FACTOR													: REAL		:= 35.4;		// Factor to convert pump percent input to rpm output (max rpm / 100)
	_BLOWER_RPM_FACTOR													: REAL      := 34.7;		// product blower rpm = 3470
	_VOLTAGE_120_FACTOR													: REAL		:= 218.44;		// 0- 150 VAC
	_VOLTAGE_240_FACTOR													: REAL		:= 65.53;		// 0 - 500 VAC 
	
	_INLET_AIR_MAX_COUNT												: INT		:= 0;
	_ADSORP_MAX_COUNT													: INT		:= 1;
	_VAC_COOLING_MAX_COUNT												: INT		:= 1;
	_DESORP_MAX_COUNT													: INT		:= 1;
	_HIGH_CART_READINGS_MAX												: INT		:= 2;
	_RETRY_ATTEMPTS														: INT		:= 3;
	_MAX_REACTOR_ERRORS													: INT		:= 3;
	
	_PRESSURE_PERCENT													: REAL		:= 0.9;
	_TEMP_DEADBAND														: REAL		:= 0.5;
	
	_TIMEOUT_WARMUP_RESET												: TIME		:= T#10M;
	_TIMEOUT_RESET														: TIME		:= T#3S;
	
	_OPEN																: INT 		:= 100;
	_CLOSED																: INT		:= 0;

	_SECONDS															: REAL		:= 1000;
	_MINUTES															: REAL		:= 60000;
	
	_U01																: STRING	:= 'U01 - ';
	_RS01																: STRING	:= 'RS01 - ';
	_R1																	: STRING	:= 'Reactor1';
	
	STEAM_TABLE  : ARRAY[1..30] OF ARRAY [0..1] OF REAL := [[0.0,0.0],[0.02,0.000015],[0.03,0.000022],[0.04,0.000029],[0.05,0.000035],[0.06,0.000042],[0.07,0.000049],[0.08,0.000055],[0.09,0.000062],
															[0.1,0.000068],[0.2,0.000131],[0.3,0.000191],[0.4,0.00025],[0.5,0.000309],[0.6,0.000366],[0.7,0.000423],[0.8,0.000479],[0.9,0.000535],
															[1.0,0.00059],[1.1,0.000645],[1.2,0.0007],[1.3,0.000755],[1.4,0.000809],[1.5,0.000863],[1.6,0.000916],[1.7,0.00097],[1.8,0.001023],[1.8,0.001023],[1.9,0.001076],
															[2.0,0.001129]];

END_VAR

// ---- GVLs/P0_Global_Variables.TcGVL
// Theseus - Global_Variables
// Rev 1.0 - October 2, 2024

VAR_GLOBAL

	gbRS01TestError														: BOOL;
	gbRS02TestError														: BOOL;
	gbRS03TestError														: BOOL;
	
	gbDrainageOn														: BOOL;
	gbCondenserKODrainageOn												: BOOL;
	gbCondensateValve													: BOOL;
	
	gbGasketsActivated													: BOOL;
	gbFirstEvacuation													: BOOL;
	giEvacuationCounter													: INT;

	gsCycleMode															: STRING;
	gsCycleStage														: STRING;
	gsM01RS01CycleStage													: STRING;
	gsM01RS02CycleStage													: STRING;
	gsM01RS03CycleStage													: STRING;
	
	gbRepresValves														: BOOL;
	
END_VAR

// ---- POUs/FB_Reactor.TcPOU
FUNCTION_BLOCK FB_Reactor
VAR_INPUT
	
	unit																: INT;

    /// <summary>XV01</summary>
	{attribute 'OPC.UA.DA' := '1'}  				                
	open_inlet_door														: BOOL;
    /// <summary>XV01</summary>
	{attribute 'OPC.UA.DA' := '1'}  				                
	close_inlet_door													: BOOL;
    /// <summary>XV03</summary>
	{attribute 'OPC.UA.DA' := '1'}  				                
	open_outlet_door													: BOOL;
    /// <summary>XV03</summary>
	{attribute 'OPC.UA.DA' := '1'}  				                
	close_outlet_door													: BOOL;

    /// <summary>XV01</summary>
	{attribute 'OPC.UA.DA' := '1'}  				                
	extend_inlet_door_clamps											: BOOL;
    /// <summary>XV01</summary>
	{attribute 'OPC.UA.DA' := '1'}  				                
	retract_inlet_door_clamps											: BOOL;
    /// <summary>XV03</summary>
	{attribute 'OPC.UA.DA' := '1'}  				                
	extend_outlet_door_clamps											: BOOL;
    /// <summary>XV03</summary>
	{attribute 'OPC.UA.DA' := '1'}  				                
	retract_outlet_door_clamps											: BOOL;

	/// <summary>XV02</summary>
	{attribute 'OPC.UA.DA' := '1'}  				                
	repres_valve														: BOOL;
	/// <summary>XV09</summary>
	{attribute 'OPC.UA.DA' := '1'}  				                
	over_pressure_test_control											: BOOL;
	
	/// <summary>AT01_pump</summary>
	{attribute 'OPC.UA.DA' := '1'}  				                
	inlet_co2_pump														: BOOL;
    /// <summary>AT01_solenoid</summary>
	{attribute 'OPC.UA.DA' := '1'}  				                
	inlet_co2_sol														: BOOL;

    /// <summary>AT03_pump</summary>
	{attribute 'OPC.UA.DA' := '1'}  				                
	outlet_co2_pump														: BOOL;
    /// <summary>AT03_solenoid</summary>
	{attribute 'OPC.UA.DA' := '1'}  				                
	outlet_co2_sol														: BOOL;
	
    /// <summary>F01</summary>
	fan_vfd_setpoint													: REAL;

END_VAR
VAR_OUTPUT

	inlet_doors_open													: BOOL;
    outlet_doors_open													: BOOL;	
    inlet_doors_closed													: BOOL;	
    outlet_doors_closed													: BOOL;	

	inlet_door_clamps_extended											: BOOL;
	inlet_door_clamps_retracted											: BOOL;
	outlet_door_clamps_extended											: BOOL;
    outlet_door_clamps_retracted										: BOOL;
	
	sorbent_low_temp													: REAL;
	sorbent_high_temp													: REAL;
	sorbent_average_temp												: REAL;

	desorption_high_temp_count											: INT;
	adsorption_high_temp_count											: INT;
	vacuum_cooling_high_temp_count										: INT;

    /// <summary>AT01</summary>																			// Summary defines hover over text while in twincat 3 program
	{attribute 'OPC.UA.DA' := '1'}  				                									// OPC_UA tag
	{attribute 'OPC.UA.DA.Access' := '1'}																// OPC_UA tag definition - '1' indicates Read Only, '2' indicates Write Only (not used), '3' indicates Read Write (default)  				                
	inlet_co2															: REAL;							// Tag value to read (scaled)
    /// <summary>AT01</summary>
	{attribute 'OPC.UA.DA' := '1'}  				                
	{attribute 'OPC.UA.DA.Access' := '1'}  				                
	inlet_co2_error														: BOOL;

    /// <summary>AT02</summary>
	{attribute 'OPC.UA.DA' := '1'}  				                
	{attribute 'OPC.UA.DA.Access' := '1'}  				                
	inlet_h2o															: REAL;
    /// <summary>AT02</summary>
	{attribute 'OPC.UA.DA' := '1'}  				                
	{attribute 'OPC.UA.DA.Access' := '1'}  				                
	inlet_h2o_error														: BOOL;

    /// <summary>AT03</summary>
	{attribute 'OPC.UA.DA' := '1'}
	{attribute 'OPC.UA.DA.Access' := '1'}  				                
	outlet_co2															: REAL;
    /// <summary>AT03</summary>
	{attribute 'OPC.UA.DA' := '1'}  				                
	{attribute 'OPC.UA.DA.Access' := '1'}  				                
	outlet_co2_error													: BOOL;

    /// <summary>AT04</summary>
	{attribute 'OPC.UA.DA' := '1'}  				                
	{attribute 'OPC.UA.DA.Access' := '1'}  				                
	outlet_h2o															: REAL;
    /// <summary>AT04</summary>
	{attribute 'OPC.UA.DA' := '1'}  				                
	{attribute 'OPC.UA.DA.Access' := '1'}  				                
	outlet_h2o_error													: BOOL;

    /// <summary>PT01</summary>
	{attribute 'OPC.UA.DA' := '1'}  				                
	{attribute 'OPC.UA.DA.Access' := '1'}  				                
	reactor_pres														: REAL;
    /// <summary>PT01</summary>
	{attribute 'OPC.UA.DA' := '1'}  				                
	{attribute 'OPC.UA.DA.Access' := '1'}  				                
	reactor_pres_error													: BOOL;

    /// <summary>FT01</summary>
	{attribute 'OPC.UA.DA' := '1'}  				                
	{attribute 'OPC.UA.DA.Access' := '1'}  				                
	air_flow															: REAL;
    /// <summary>FT01</summary>
	{attribute 'OPC.UA.DA' := '1'}  				                
	{attribute 'OPC.UA.DA.Access' := '1'}  				                
	air_flow_error														: BOOL;

    /// <summary>PDT01</summary>
	{attribute 'OPC.UA.DA' := '1'}  				                
	{attribute 'OPC.UA.DA.Access' := '1'}  				                
	filter_diff_pres													: REAL;
    /// <summary>PDT01</summary>
	{attribute 'OPC.UA.DA' := '1'}  				                
	{attribute 'OPC.UA.DA.Access' := '1'}  				                
	filter_diff_pres_error												: BOOL;

    /// <summary>PDT02</summary>
	{attribute 'OPC.UA.DA' := '1'}  				                
	{attribute 'OPC.UA.DA.Access' := '1'}  				                
	sorbent_diff_pres													: REAL;
    /// <summary>PDT02</summary>
	{attribute 'OPC.UA.DA' := '1'}  				                
	{attribute 'OPC.UA.DA.Access' := '1'}  				                
	sorbent_diff_pres_error												: BOOL;

    /// <summary>PDT03</summary>
	{attribute 'OPC.UA.DA' := '1'}  				                
	{attribute 'OPC.UA.DA.Access' := '1'}  				                
	fan_diff_pres														: REAL;
    /// <summary>PDT03</summary>
	{attribute 'OPC.UA.DA' := '1'}  				                
	{attribute 'OPC.UA.DA.Access' := '1'}  				                
	fan_diff_pres_error													: BOOL;
    /// <summary>TT04</summary>
	{attribute 'OPC.UA.DA' := '1'}  				                
	{attribute 'OPC.UA.DA.Access' := '1'}  				                
	air_inlet_temp														: REAL;
    /// <summary>TT04</summary>
	{attribute 'OPC.UA.DA' := '1'}  				                
	{attribute 'OPC.UA.DA.Access' := '1'}  				                
	air_inlet_temp_error												: BOOL;
	
    /// <summary>TT05</summary>
	{attribute 'OPC.UA.DA' := '1'}  				                
	{attribute 'OPC.UA.DA.Access' := '1'}  				                
	reactor_wall_temp													: REAL;
    /// <summary>Reactor Wall Temp</summary>
	{attribute 'OPC.UA.DA' := '1'}  				                
	{attribute 'OPC.UA.DA.Access' := '1'}  				                
	reactor_wall_temp_error												: BOOL;
	
    /// <summary>AT01_pump</summary>
	{attribute 'OPC.UA.DA' := '1'}  				                
	{attribute 'OPC.UA.DA.Access' := '1'}  				                
	inlet_co2_pump_cmd_status											: BOOL;
    /// <summary>AT01_solenoid</summary>
	{attribute 'OPC.UA.DA' := '1'}  				                
	{attribute 'OPC.UA.DA.Access' := '1'}  				                
	inlet_co2_sol_cmd_status											: BOOL;

    /// <summary>AT03_pump</summary>
	{attribute 'OPC.UA.DA' := '1'}  				                
	{attribute 'OPC.UA.DA.Access' := '1'}  				                
	outlet_co2_pump_cmd_status											: BOOL;
    /// <summary>AT03_solenoid</summary>
	{attribute 'OPC.UA.DA' := '1'}  				                
	{attribute 'OPC.UA.DA.Access' := '1'}  				                
	outlet_co2_sol_cmd_status											: BOOL;
	
    /// <summary>XV-02</summary>
	repres_valve_clear													: BOOL;

    /// <summary>XV09</summary>
	{attribute 'OPC.UA.DA' := '1'}  				                
	{attribute 'OPC.UA.DA.Access' := '1'}  				                
	over_pressure_test_control_cmd_status								: BOOL;

END_VAR
VAR
	fb_Fan																: FB_VFD();
	tonFan																: TON;
	rRpm																: REAL;
	rFanSPOld															: REAL			:= 0;

	fbInletDoorsClosed													: FB_Door_Closed();
	fbOutletDoorsClosed													: FB_Door_Closed();
	
	rtrigSorbentErrorCheck												: R_TRIG;
	i																	: INT;
	iCount																: ARRAY [0..23] OF INT;

	iInletAirSetpoint													: INT			:= 0;
	iTempCount															: INT;
	iHighTempCount														: INT;
	rTempTotal															: REAL;
	rTempSP																: REAL;
	rMin																: REAL;
	rMax																: REAL;

	cart01_temp_front_calc												: FB_Temperature;
	cart01_temp_back_calc												: FB_Temperature;
	cart02_temp_front_calc												: FB_Temperature;
	cart02_temp_back_calc												: FB_Temperature;
	cart03_temp_front_calc												: FB_Temperature;
	cart03_temp_back_calc												: FB_Temperature;
	cart04_temp_front_calc												: FB_Temperature;
	cart04_temp_back_calc												: FB_Temperature;
	cart05_temp_front_calc												: FB_Temperature;
	cart05_temp_back_calc												: FB_Temperature;
	cart06_temp_front_calc												: FB_Temperature;
	cart06_temp_back_calc												: FB_Temperature;
	cart07_temp_front_calc												: FB_Temperature;
	cart07_temp_back_calc												: FB_Temperature;
	cart08_temp_front_calc												: FB_Temperature;
	cart08_temp_back_calc												: FB_Temperature;
	cart09_temp_front_calc												: FB_Temperature;
	cart09_temp_back_calc												: FB_Temperature;
	cart10_temp_front_calc												: FB_Temperature;
	cart10_temp_back_calc												: FB_Temperature;
	cart11_temp_front_calc												: FB_Temperature;
	cart11_temp_back_calc												: FB_Temperature;
	cart12_temp_front_calc												: FB_Temperature;
	cart12_temp_back_calc												: FB_Temperature;
	
    /// <summary>AT01</summary>
	{attribute 'OPC.UA.DA' := '1'}  				                
	_InletCO2ErrorOff													: BOOL;
    /// <summary>Inlet CO2</summary>
	AT_01														AT %I*	: INT;
    /// <summary>Inlet CO2</summary>
	{attribute 'OPC.UA.DA' := '1'}
	{attribute 'OPC.UA.DA.Access' := '1'}  				                
	AT_01_error													AT %I*	: BOOL;

    /// <summary>AT02</summary>
	{attribute 'OPC.UA.DA' := '1'}  				                
	_InletH2OErrorOff													: BOOL;
    /// <summary>Inlet H20</summary>
	AT_02														AT %I*	: INT;
    /// <summary>Inlet H20</summary>
	{attribute 'OPC.UA.DA' := '1'}  				                
	{attribute 'OPC.UA.DA.Access' := '1'}  				                
	AT_02_error													AT %I*	: BOOL;

    /// <summary>AT03</summary>
	{attribute 'OPC.UA.DA' := '1'}  				                
	_OutletCO2ErrorOff													: BOOL;
    /// <summary>Outlet CO2</summary>
	AT_03														AT %I*	: INT;
    /// <summary>Outlet CO2</summary>
	{attribute 'OPC.UA.DA' := '1'}
	{attribute 'OPC.UA.DA.Access' := '1'}  				                
	AT_03_error													AT %I*	: BOOL;

    /// <summary>AT04</summary>
	{attribute 'OPC.UA.DA' := '1'}  				                
	_OutletH2OErrorOff													: BOOL;
    /// <summary>Outlet H20</summary>
	AT_04														AT %I*	: INT;
    /// <summary>Outlet H20</summary>
	{attribute 'OPC.UA.DA' := '1'}  				                
	{attribute 'OPC.UA.DA.Access' := '1'}  				                
	AT_04_error													AT %I*	: BOOL;

    /// <summary>PT01</summary>
	{attribute 'OPC.UA.DA' := '1'}
	_ReactorPresErrorOff												: BOOL;  				                
    /// <summary>Reactor Pressure</summary>
	PT_01														AT %I*	: INT;
    /// <summary>Reactor Pressure</summary>
	{attribute 'OPC.UA.DA' := '1'}  				                
	{attribute 'OPC.UA.DA.Access' := '1'}  				                
	PT_01_error													AT %I*	: BOOL;

    /// <summary>FT01</summary>
	{attribute 'OPC.UA.DA' := '1'}  				                
	_AirFlowErrorOff													: BOOL;
    /// <summary>Air flow</summary>
	FT_01														AT %I*	: INT;
    /// <summary>Air flow</summary>
	{attribute 'OPC.UA.DA' := '1'}  				                
	{attribute 'OPC.UA.DA.Access' := '1'}  				                
	FT_01_error													AT %I*	: BOOL;

    /// <summary>PDT01</summary>
	{attribute 'OPC.UA.DA' := '1'}  				                
	_FilterDiffPresErrorOff												: BOOL;
    /// <summary>Filter diff pres</summary>
	PDT_01														AT %I*	: INT;
    /// <summary>Filter diff pres</summary>
	{attribute 'OPC.UA.DA' := '1'}  				                
	{attribute 'OPC.UA.DA.Access' := '1'}  				                
	PDT_01_error												AT %I*	: BOOL;

    /// <summary>PDT02</summary>
	{attribute 'OPC.UA.DA' := '1'}  				                
	_SorbentDiffPresErrorOff											: BOOL;
    /// <summary>Sorbent diff pres</summary>
	PDT_02														AT %I*	: INT;
    /// <summary>Sorbent diff pres</summary>
	{attribute 'OPC.UA.DA' := '1'}  				                
	{attribute 'OPC.UA.DA.Access' := '1'}  				                
	PDT_02_error												AT %I*	: BOOL;

    /// <summary>PDT03</summary>
	{attribute 'OPC.UA.DA' := '1'}  				                
	_FanDiffPresErrorOff												: BOOL;
    /// <summary>fan diff pres</summary>
	PDT_03														AT %I*	: INT;
    /// <summary>fan diff pres</summary>
	{attribute 'OPC.UA.DA' := '1'}  				                
	{attribute 'OPC.UA.DA.Access' := '1'}  				                
	PDT_03_error												AT %I*	: BOOL;
	
    /// <summary>TT04</summary>
	{attribute 'OPC.UA.DA' := '1'}  				                
	_AirInletTempErrorOff												: BOOL;
    /// <summary>air inlet temp</summary>
	TT_04														AT %I*	: INT;
    /// <summary>air inlet temp</summary>
	{attribute 'OPC.UA.DA' := '1'}  				                
	{attribute 'OPC.UA.DA.Access' := '1'}  				                
	TT_04_error													AT %I*	: BOOL;

    /// <summary>TT05</summary>
	_ReactorWallTempErrorOff											: BOOL;
    /// <summary>Reactor wall temp</summary>
	TT_05														AT %I*	: INT;
    /// <summary>Reactor wall temp</summary>
	{attribute 'OPC.UA.DA' := '1'}  				                
	{attribute 'OPC.UA.DA.Access' := '1'}  				                
	TT_05_error													AT %I*	: BOOL;
	
    /// <summary>Inlet CO2 pump</summary>
	AT_01_pump													AT %Q*	: BOOL;
    /// <summary>Inlet CO2 solenoid</summary>
	AT_01_sol													AT %Q*	: BOOL;

    /// <summary>Inlet CO2 pump</summary>
	AT_03_pump													AT %Q*	: BOOL;
    /// <summary>Outlet CO2 solenoid</summary>
	AT_03_sol													AT %Q*	: BOOL;

    /// <summary>XV02</summary>
	{attribute 'OPC.UA.DA' := '1'}  				                
	{attribute 'OPC.UA.DA.Access' := '1'}  				                
	repres_valve_open_cmd_status										: BOOL;
    /// <summary>XV02</summary>
	{attribute 'OPC.UA.DA' := '1'}  				                
	{attribute 'OPC.UA.DA.Access' := '1'}  				                
	repres_valve_open											AT %I*	: BOOL;
    /// <summary>XV02</summary>
	{attribute 'OPC.UA.DA' := '1'}  				                
	{attribute 'OPC.UA.DA.Access' := '1'}  				                
	repres_valve_closed											AT %I*	: BOOL;
    /// <summary>repres valve</summary>
	XV_02														AT %Q*	: BOOL;
	
    /// <summary>over pressure test control</summary>
	XV_09														AT %Q*	: BOOL;
	
    /// <summary>F01</summary>
	{attribute 'OPC.UA.DA' := '1'}  				                
	fan_vfd_enable														: BOOL :=  TRUE;
    /// <summary>F01</summary>
	{attribute 'OPC.UA.DA' := '1'}  				                
	fan_vfd_reset														: BOOL;
    /// <summary>F01</summary>
	{attribute 'OPC.UA.DA' := '1'}  				                
	{attribute 'OPC.UA.DA.Access' := '1'}  				                
	fan_vfd_enabled														: BOOL;
    /// <summary>F01</summary>
	{attribute 'OPC.UA.DA' := '1'}  				                
	{attribute 'OPC.UA.DA.Access' := '1'}  				                
	fan_vfd_error														: BOOL;
    /// <summary>F01</summary>
	{attribute 'OPC.UA.DA' := '1'}  				                
	{attribute 'OPC.UA.DA.Access' := '1'}  				                
	fan_vfd_output														: REAL;
	 /// <summary>F01</summary>
	{attribute 'OPC.UA.DA' := '1'}  				                
	{attribute 'OPC.UA.DA.Access' := '1'}  				                
	fan_vfd_output_current												: REAL;
    /// <summary>F01</summary>
	fan_vfd_control												AT %Q*	: WORD;
    /// <summary>F01</summary>
	fan_vfd_target_vel											AT %Q*	: WORD;
    /// <summary>F01</summary>
	fan_vfd_status												AT %I*	: WORD;
    /// <summary>F01</summary>
	fan_vfd_velocity											AT %I*	: WORD;
    /// <summary>F01</summary>
	fan_vfd_ecat_state											AT %I*  : BOOL;
	fan_vfd_current												AT %I*	: DINT;
	//fan_vfd_current_amps										AT %Q*	: REAL;

    /// <summary>XV01_SV05</summary>
	inlet_door_open_valve										AT %Q*	: BOOL;
    /// <summary>XV01_SV06</summary>
	inlet_door_close_valve										AT %Q*	: BOOL;
	
    /// <summary>XV01_ZS01</summary>
	{attribute 'OPC.UA.DA' := '1'}  				                
	{attribute 'OPC.UA.DA.Access' := '1'}  				                
	inlet_door_near_open_ls										AT %I*	: BOOL;
    /// <summary>XV01_ZS02</summary>
	{attribute 'OPC.UA.DA' := '1'}  				                
	{attribute 'OPC.UA.DA.Access' := '1'}  				                
	inlet_door_near_closed_ls									AT %I*	: BOOL;
    /// <summary>XV01_ZS02</summary>
	{attribute 'OPC.UA.DA' := '1'}  				                
	{attribute 'OPC.UA.DA.Access' := '1'}  				                
	inlet_door_near_closed												: BOOL;
    /// <summary>XV01_ZS04</summary>
	{attribute 'OPC.UA.DA' := '1'}  				                
	{attribute 'OPC.UA.DA.Access' := '1'}  				                
	inlet_door_far_open_ls										AT %I*	: BOOL;
    /// <summary>XV01_ZS05</summary>
	{attribute 'OPC.UA.DA' := '1'}  				                
	{attribute 'OPC.UA.DA.Access' := '1'}  				                
	inlet_door_far_closed_ls									AT %I*	: BOOL;
    /// <summary>XV01_ZS05</summary>
	{attribute 'OPC.UA.DA' := '1'}  				                
	{attribute 'OPC.UA.DA.Access' := '1'}  				                
	inlet_door_far_closed												: BOOL;
	
    /// <summary>XV01_ZS03</summary>
	{attribute 'OPC.UA.DA' := '1'}  				                
	{attribute 'OPC.UA.DA.Access' := '1'}  				                
	inlet_door_near_clamps_extended								AT %I*	: BOOL;
    /// <summary>XV01_ZS06</summary>
	{attribute 'OPC.UA.DA' := '1'}  				                
	{attribute 'OPC.UA.DA.Access' := '1'}  				                
	inlet_door_far_clamps_extended								AT %I*	: BOOL;

    /// <summary>XV01_SV01</summary>
	inlet_door_near_clamps_extend_valve							AT %Q*	: BOOL;
    /// <summary>XV01_SV03</summary>
	inlet_door_near_clamps_retract_valve						AT %Q*	: BOOL;
    /// <summary>XV01_SV02 Clamps</summary>
	inlet_door_far_clamps_extend_valve							AT %Q*	: BOOL;
    /// <summary>XV01_SV04</summary>
	inlet_door_far_clamps_retract_valve							AT %Q*	: BOOL;

    /// <summary>XV03_SV05</summary>
	outlet_door_open_valve										AT %Q*	: BOOL;
    /// <summary>XV03_SV06</summary>
	outlet_door_close_valve										AT %Q*	: BOOL;

    /// <summary>XV03 ZS01</summary>
	{attribute 'OPC.UA.DA' := '1'}  				                
	{attribute 'OPC.UA.DA.Access' := '1'}  				                
	outlet_door_near_open_ls									AT %I*	: BOOL;
    /// <summary>XV03 ZS02</summary>
	{attribute 'OPC.UA.DA' := '1'}  				                
	{attribute 'OPC.UA.DA.Access' := '1'}  				                
	outlet_door_near_closed_ls									AT %I*	: BOOL;
    /// <summary>XV03 ZS02</summary>
	{attribute 'OPC.UA.DA' := '1'}  				                
	{attribute 'OPC.UA.DA.Access' := '1'}  				                
	outlet_door_near_closed												: BOOL;
    /// <summary>XV03 ZS04</summary>
	{attribute 'OPC.UA.DA' := '1'}  				                
	{attribute 'OPC.UA.DA.Access' := '1'}  				                
	outlet_door_far_open_ls										AT %I*	: BOOL;
    /// <summary>XV03 ZS05</summary>
	{attribute 'OPC.UA.DA' := '1'}  				                
	{attribute 'OPC.UA.DA.Access' := '1'}  				                
	outlet_door_far_closed_ls									AT %I*	: BOOL;
    /// <summary>XV03 ZS05</summary>
	{attribute 'OPC.UA.DA' := '1'}  				                
	{attribute 'OPC.UA.DA.Access' := '1'}  				                
	outlet_door_far_closed												: BOOL;

    /// <summary>XV03 ZS03</summary>
	{attribute 'OPC.UA.DA' := '1'}  				                
	{attribute 'OPC.UA.DA.Access' := '1'}  				                
	outlet_door_near_clamps_extended							AT %I*	: BOOL;
    /// <summary>XV03 ZS06</summary>
	{attribute 'OPC.UA.DA' := '1'}  				                
	{attribute 'OPC.UA.DA.Access' := '1'}  				                
	outlet_door_far_clamps_extended								AT %I*	: BOOL;
	
    /// <summary>XV03_SV01</summary>
	outlet_door_near_clamps_extend_valve						AT %Q*	: BOOL;
    /// <summary>XV03_SV03</summary>
	outlet_door_near_clamps_retract_valve						AT %Q*	: BOOL;
    /// <summary>XV03_SV02</summary>
	outlet_door_far_clamps_extend_valve							AT %Q*	: BOOL;
    /// <summary>XV03_SV04</summary>
	outlet_door_far_clamps_retract_valve						AT %Q*	: BOOL;

   /// <summary>01-TT-01</summary>
	{attribute 'OPC.UA.DA' := '1'}  				                
	{attribute 'OPC.UA.DA.Access' := '1'}  				                
	cart01_front_temp													: REAL;
    /// <summary>01-TT-01</summary>
	{attribute 'OPC.UA.DA' := '1'}  				                
	{attribute 'OPC.UA.DA.Access' := '1'}  				                
	cart01_front_temp_error												: BOOL;
    /// <summary>Cart01 front temperature</summary>
	_01_TT_01													AT %I*	: INT;
    /// <summary>Cart01 front temperature</summary>
	_01_TT_01_Error												AT %I*	: BOOL;

    /// <summary>01-TT-03</summary>
	{attribute 'OPC.UA.DA' := '1'}  				                
	{attribute 'OPC.UA.DA.Access' := '1'}  				                
	cart01_back_temp													: REAL;
    /// <summary>01-TT-03</summary>
	{attribute 'OPC.UA.DA' := '1'}  				                
	{attribute 'OPC.UA.DA.Access' := '1'}  				                
	cart01_back_temp_error												: BOOL;
    /// <summary>Cart01 back temperature</summary>
	_01_TT_03													AT %I*	: INT;
    /// <summary>Cart01 back temperature</summary>
	_01_TT_03_Error												AT %I*	: BOOL;
	
    /// <summary>02-TT-01</summary>
	{attribute 'OPC.UA.DA' := '1'}  				                
	{attribute 'OPC.UA.DA.Access' := '1'}  				                
	cart02_front_temp													: REAL;
    /// <summary>02-TT-01</summary>
	{attribute 'OPC.UA.DA' := '1'}  				                
	{attribute 'OPC.UA.DA.Access' := '1'}  				                
	cart02_front_temp_error												: BOOL;
    /// <summary>Cart02 front temperature</summary>
	_02_TT_01													AT %I*	: INT;
    /// <summary>Cart02 front temperature</summary>
	_02_TT_01_Error												AT %I*	: BOOL;

    /// <summary>02-TT-03</summary>
	{attribute 'OPC.UA.DA' := '1'}  				                
	{attribute 'OPC.UA.DA.Access' := '1'}  				                
	cart02_back_temp													: REAL;
    /// <summary>02-TT-03</summary>
	{attribute 'OPC.UA.DA' := '1'}  				                
	{attribute 'OPC.UA.DA.Access' := '1'}  				                
	cart02_back_temp_error												: BOOL;
    /// <summary>Cart02 back temperature</summary>
	_02_TT_03													AT %I*	: INT;
    /// <summary>Cart02 back temperature</summary>
	_02_TT_03_Error												AT %I*	: BOOL;
	
    /// <summary>03-TT-01</summary>
	{attribute 'OPC.UA.DA' := '1'}  				                
	{attribute 'OPC.UA.DA.Access' := '1'}  				                
	cart03_front_temp													: REAL;
    /// <summary>03-TT-01</summary>
	{attribute 'OPC.UA.DA' := '1'}  				                
	{attribute 'OPC.UA.DA.Access' := '1'}  				                
	cart03_front_temp_error												: BOOL;
    /// <summary>Cart03 front temperature</summary>
	_03_TT_01													AT %I*	: INT;
    /// <summary>Cart03 front temperature</summary>
	_03_TT_01_Error												AT %I*	: BOOL;

    /// <summary>03-TT-03</summary>
	{attribute 'OPC.UA.DA' := '1'}  				                
	{attribute 'OPC.UA.DA.Access' := '1'}  				                
	cart03_back_temp													: REAL;
    /// <summary>03-TT-03</summary>
	{attribute 'OPC.UA.DA' := '1'}  				                
	{attribute 'OPC.UA.DA.Access' := '1'}  				                
	cart03_back_temp_error												: BOOL;
    /// <summary>Cart03 back temperature</summary>
	_03_TT_03													AT %I*	: INT;
    /// <summary>Cart03 back temperature</summary>
	_03_TT_03_Error												AT %I*	: BOOL;

    /// <summary>04-TT-01</summary>
	{attribute 'OPC.UA.DA' := '1'}  				                
	{attribute 'OPC.UA.DA.Access' := '1'}  				                
	cart04_front_temp													: REAL;
    /// <summary>04-TT-01</summary>
	{attribute 'OPC.UA.DA' := '1'}  				                
	{attribute 'OPC.UA.DA.Access' := '1'}  				                
	cart04_front_temp_error												: BOOL;
    /// <summary>Cart04 front temperature</summary>
	_04_TT_01													AT %I*	: INT;
    /// <summary>Cart04 front temperature</summary>
	_04_TT_01_Error												AT %I*	: BOOL;

    /// <summary>04-TT-03</summary>
	{attribute 'OPC.UA.DA' := '1'}  				                
	{attribute 'OPC.UA.DA.Access' := '1'}  				                
	cart04_back_temp													: REAL;
    /// <summary>04-TT-03</summary>
	{attribute 'OPC.UA.DA' := '1'}  				                
	{attribute 'OPC.UA.DA.Access' := '1'}  				                
	cart04_back_temp_error												: BOOL;
    /// <summary>Cart04 back temperature</summary>
	_04_TT_03													AT %I*	: INT;
    /// <summary>Cart04 back temperature</summary>
	_04_TT_03_Error												AT %I*	: BOOL;

    /// <summary>05-TT-01</summary>
	{attribute 'OPC.UA.DA' := '1'}  				                
	{attribute 'OPC.UA.DA.Access' := '1'}  				                
	cart05_front_temp													: REAL;
    /// <summary>05-TT-01</summary>
	{attribute 'OPC.UA.DA' := '1'}  				                
	{attribute 'OPC.UA.DA.Access' := '1'}  				                
	cart05_front_temp_error												: BOOL;
    /// <summary>Cart05 front temperature</summary>
	_05_TT_01													AT %I*	: INT;
    /// <summary>Cart05 front temperature</summary>
	_05_TT_01_Error												AT %I*	: BOOL;

    /// <summary>05-TT-03</summary>
	{attribute 'OPC.UA.DA' := '1'}  				                
	{attribute 'OPC.UA.DA.Access' := '1'}  				                
	cart05_back_temp													: REAL;
    /// <summary>05-TT-03</summary>
	{attribute 'OPC.UA.DA' := '1'}  				                
	{attribute 'OPC.UA.DA.Access' := '1'}  				                
	cart05_back_temp_error												: BOOL;
    /// <summary>Cart05 back temperature</summary>
	_05_TT_03													AT %I*	: INT;
    /// <summary>Cart05 back temperature</summary>
	_05_TT_03_Error												AT %I*	: BOOL;
	
    /// <summary>06-TT-01</summary>
	{attribute 'OPC.UA.DA' := '1'}  				                
	{attribute 'OPC.UA.DA.Access' := '1'}  				                
	cart06_front_temp													: REAL;
    /// <summary>06-TT-01</summary>
	{attribute 'OPC.UA.DA' := '1'}  				                
	{attribute 'OPC.UA.DA.Access' := '1'}  				                
	cart06_front_temp_error												: BOOL;
    /// <summary>Cart06 front temperature</summary>
	_06_TT_01													AT %I*	: INT;
    /// <summary>Cart06 front temperature</summary>
	_06_TT_01_Error												AT %I*	: BOOL;

    /// <summary>06-TT-03</summary>
	{attribute 'OPC.UA.DA' := '1'}  				                
	{attribute 'OPC.UA.DA.Access' := '1'}  				                
	cart06_back_temp													: REAL;
    /// <summary>06-TT-03</summary>
	{attribute 'OPC.UA.DA' := '1'}  				                
	{attribute 'OPC.UA.DA.Access' := '1'}  				                
	cart06_back_temp_error												: BOOL;
    /// <summary>Cart06 back temperature</summary>
	_06_TT_03													AT %I*	: INT;
    /// <summary>Cart06 back temperature</summary>
	_06_TT_03_Error												AT %I*	: BOOL;
	
    /// <summary>07-TT-01</summary>
	{attribute 'OPC.UA.DA' := '1'}  				                
	{attribute 'OPC.UA.DA.Access' := '1'}  				                
	cart07_front_temp													: REAL;
    /// <summary>07-TT-01</summary>
	{attribute 'OPC.UA.DA' := '1'}  				                
	{attribute 'OPC.UA.DA.Access' := '1'}  				                
	cart07_front_temp_error												: BOOL;
    /// <summary>Cart07 front temperature</summary>
	_07_TT_01													AT %I*	: INT;
    /// <summary>Cart07 front temperature</summary>
	_07_TT_01_Error												AT %I*	: BOOL;

    /// <summary>07-TT-03</summary>
	{attribute 'OPC.UA.DA' := '1'}  				                
	{attribute 'OPC.UA.DA.Access' := '1'}  				                
	cart07_back_temp													: REAL;
    /// <summary>07-TT-03</summary>
	{attribute 'OPC.UA.DA' := '1'}  				                
	{attribute 'OPC.UA.DA.Access' := '1'}  				                
	cart07_back_temp_error												: BOOL;
    /// <summary>Cart07 back temperature</summary>
	_07_TT_03													AT %I*	: INT;
    /// <summary>Cart07 back temperature</summary>
	_07_TT_03_Error												AT %I*	: BOOL;
	
    /// <summary>08-TT-01</summary>
	{attribute 'OPC.UA.DA' := '1'}  				                
	{attribute 'OPC.UA.DA.Access' := '1'}  				                
	cart08_front_temp													: REAL;
    /// <summary>08-TT-01</summary>
	{attribute 'OPC.UA.DA' := '1'}  				                
	{attribute 'OPC.UA.DA.Access' := '1'}  				                
	cart08_front_temp_error												: BOOL;
    /// <summary>Cart08 front temperature</summary>
	_08_TT_01													AT %I*	: INT;
    /// <summary>Cart08 front temperature</summary>
	_08_TT_01_Error												AT %I*	: BOOL;

    /// <summary>08-TT-03</summary>
	{attribute 'OPC.UA.DA' := '1'}  				                
	{attribute 'OPC.UA.DA.Access' := '1'}  				                
	cart08_back_temp													: REAL;
    /// <summary>08-TT-03</summary>
	{attribute 'OPC.UA.DA' := '1'}  				                
	{attribute 'OPC.UA.DA.Access' := '1'}  				                
	cart08_back_temp_error												: BOOL;
    /// <summary>Cart08 back temperature</summary>
	_08_TT_03													AT %I*	: INT;
    /// <summary>Cart08 back temperature</summary>
	_08_TT_03_Error												AT %I*	: BOOL;
	
    /// <summary>09-TT-01</summary>
	{attribute 'OPC.UA.DA' := '1'}  				                
	{attribute 'OPC.UA.DA.Access' := '1'}  				                
	cart09_front_temp													: REAL;
    /// <summary>09-TT-01</summary>
	{attribute 'OPC.UA.DA' := '1'}  				                
	{attribute 'OPC.UA.DA.Access' := '1'}  				                
	cart09_front_temp_error												: BOOL;
    /// <summary>Cart09 front temperature</summary>
	_09_TT_01													AT %I*	: INT;
    /// <summary>Cart09 front temperature</summary>
	_09_TT_01_Error												AT %I*	: BOOL;

    /// <summary>09-TT-03</summary>
	{attribute 'OPC.UA.DA' := '1'}  				                
	{attribute 'OPC.UA.DA.Access' := '1'}  				                
	cart09_back_temp													: REAL;
    /// <summary>09-TT-03</summary>
	{attribute 'OPC.UA.DA' := '1'}  				                
	{attribute 'OPC.UA.DA.Access' := '1'}  				                
	cart09_back_temp_error												: BOOL;
    /// <summary>Cart09 back temperature</summary>
	_09_TT_03													AT %I*	: INT;
    /// <summary>Cart09 back temperature</summary>
	_09_TT_03_Error												AT %I*	: BOOL;
	
    /// <summary>10-TT-01</summary>
	{attribute 'OPC.UA.DA' := '1'}  				                
	{attribute 'OPC.UA.DA.Access' := '1'}  				                
	cart10_front_temp													: REAL;
    /// <summary>10-TT-01</summary>
	{attribute 'OPC.UA.DA' := '1'}  				                
	{attribute 'OPC.UA.DA.Access' := '1'}  				                
	cart10_front_temp_error												: BOOL;
    /// <summary>Cart10 front temperature</summary>
	_10_TT_01													AT %I*	: INT;
    /// <summary>Cart10 front temperature</summary>
	_10_TT_01_Error												AT %I*	: BOOL;

    /// <summary>10-TT-03</summary>
	{attribute 'OPC.UA.DA' := '1'}  				                
	{attribute 'OPC.UA.DA.Access' := '1'}  				                
	cart10_back_temp													: REAL;
    /// <summary>10-TT-03</summary>
	{attribute 'OPC.UA.DA' := '1'}  				                
	{attribute 'OPC.UA.DA.Access' := '1'}  				                
	cart10_back_temp_error												: BOOL;
    /// <summary>Cart10 back temperature</summary>
	_10_TT_03													AT %I*	: INT;
    /// <summary>Cart10 back temperature</summary>
	_10_TT_03_Error												AT %I*	: BOOL;

    /// <summary>11-TT-01</summary>
	{attribute 'OPC.UA.DA' := '1'}  				                
	{attribute 'OPC.UA.DA.Access' := '1'}  				                
	cart11_front_temp													: REAL;
    /// <summary>11-TT-01</summary>
	{attribute 'OPC.UA.DA' := '1'}  				                
	{attribute 'OPC.UA.DA.Access' := '1'}  				                
	cart11_front_temp_error												: BOOL;
    /// <summary>Cart11 front temperature</summary>
	_11_TT_01													AT %I*	: INT;
    /// <summary>Cart11 front temperature</summary>
	_11_TT_01_Error												AT %I*	: BOOL;

    /// <summary>11-TT-03</summary>
	{attribute 'OPC.UA.DA' := '1'}  				                
	{attribute 'OPC.UA.DA.Access' := '1'}  				                
	cart11_back_temp													: REAL;
    /// <summary>11-TT-03</summary>
	{attribute 'OPC.UA.DA' := '1'}  				                
	{attribute 'OPC.UA.DA.Access' := '1'}  				                
	cart11_back_temp_error												: BOOL;
    /// <summary>Cart11 back temperature</summary>
	_11_TT_03													AT %I*	: INT;
    /// <summary>Cart11 back temperature</summary>
	_11_TT_03_Error												AT %I*	: BOOL;

    /// <summary>12-TT-01</summary>
	{attribute 'OPC.UA.DA' := '1'}  				                
	{attribute 'OPC.UA.DA.Access' := '1'}  				                
	cart12_front_temp													: REAL;
    /// <summary>12-TT-01</summary>
	{attribute 'OPC.UA.DA' := '1'}  				                
	{attribute 'OPC.UA.DA.Access' := '1'}  				                
	cart12_front_temp_error												: BOOL;
    /// <summary>Cart12 front temperature</summary>
	_12_TT_01													AT %I*	: INT;
    /// <summary>Cart12 front temperature</summary>
	_12_TT_01_Error												AT %I*	: BOOL;

    /// <summary>12-TT-03</summary>
	{attribute 'OPC.UA.DA' := '1'}  				                
	{attribute 'OPC.UA.DA.Access' := '1'}  				                
	cart12_back_temp													: REAL;
    /// <summary>12-TT-03</summary>
	{attribute 'OPC.UA.DA' := '1'}  				                
	{attribute 'OPC.UA.DA.Access' := '1'}  				                
	cart12_back_temp_error												: BOOL;
    /// <summary>Cart12 back temperature</summary>
	_12_TT_03													AT %I*	: INT;
    /// <summary>Cart12 back temperature</summary>
	_12_TT_03_Error												AT %I*	: BOOL;
	
	{attribute 'OPC.UA.DA' := '1'}  				                
	{attribute 'OPC.UA.DA.Access' := '1'}  				                
	temp_low															: REAL;
	{attribute 'OPC.UA.DA' := '1'}  				                
	{attribute 'OPC.UA.DA.Access' := '1'}  				                
	temp_high															: REAL;
	{attribute 'OPC.UA.DA' := '1'}  				                
	{attribute 'OPC.UA.DA.Access' := '1'}  				                
	temp_average														: REAL;

END_VAR

VAR PERSISTENT

    /// <summary>AT-01</summary>
	{attribute 'OPC.UA.DA' := '1'}  				                
	inlet_co2_low														: REAL;							// Tag for low point to scale input (these tags can be preset as shown or overwritten)
    /// <summary>AT-01</summary>
	{attribute 'OPC.UA.DA' := '1'}  				                
	inlet_co2_high														: REAL;							// Tag for high point to scale input
    /// <summary>AT-01</summary>
	{attribute 'OPC.UA.DA' := '1'}  				                
	inlet_co2_min														: REAL;							// Tag for minimum display value (if input is below this value, zero is displayed)
    /// <summary>AT-01</summary>
	{attribute 'OPC.UA.DA' := '1'}  				                
	inlet_co2_offset													: REAL;							// Tag for offset correction value

    /// <summary>AT-02</summary>
	{attribute 'OPC.UA.DA' := '1'}  				                
	inlet_h2o_low														: REAL;
    /// <summary>AT-02</summary>
	{attribute 'OPC.UA.DA' := '1'}  				                
	inlet_h2o_high														: REAL;
    /// <summary>AT-02</summary>
	{attribute 'OPC.UA.DA' := '1'}  				                
	inlet_h2o_min														: REAL;
    /// <summary>AT-02</summary>
	{attribute 'OPC.UA.DA' := '1'}  				                
	inlet_h2o_offset													: REAL;

    /// <summary>AT-03</summary>
	{attribute 'OPC.UA.DA' := '1'}  				                
	outlet_co2_low														: REAL;
    /// <summary>AT-03</summary>
	{attribute 'OPC.UA.DA' := '1'}  				                
	outlet_co2_high														: REAL;
    /// <summary>AT-03</summary>
	{attribute 'OPC.UA.DA' := '1'}  				                
	outlet_co2_min														: REAL;
    /// <summary>AT-03</summary>
	{attribute 'OPC.UA.DA' := '1'}  				                
	outlet_co2_offset													: REAL;

    /// <summary>AT-04</summary>
	{attribute 'OPC.UA.DA' := '1'}  				                
	outlet_h2o_low														: REAL;
    /// <summary>AT-04</summary>
	{attribute 'OPC.UA.DA' := '1'}  				                
	outlet_h2o_high														: REAL;
    /// <summary>AT-04</summary>
	{attribute 'OPC.UA.DA' := '1'}  				                
	outlet_h2o_min														: REAL;
    /// <summary>AT-04</summary>
	{attribute 'OPC.UA.DA' := '1'}  				                
	outlet_h2o_offset													: REAL;
	
    /// <summary>FT01</summary>
	{attribute 'OPC.UA.DA' := '1'}  				                
	air_flow_low														: REAL;
    /// <summary>FT01</summary>
	{attribute 'OPC.UA.DA' := '1'}  				                
	air_flow_high														: REAL;
    /// <summary>FT01</summary>
	{attribute 'OPC.UA.DA' := '1'}  				                
	air_flow_min														: REAL;
    /// <summary>FT01</summary>
	{attribute 'OPC.UA.DA' := '1'}  				                
	air_flow_offset														: REAL;

    /// <summary>PDT-01</summary>
	{attribute 'OPC.UA.DA' := '1'}  				                
	filter_diff_pres_low												: REAL;
    /// <summary>PDT-01</summary>
	{attribute 'OPC.UA.DA' := '1'}  				                
	filter_diff_pres_high												: REAL;
    /// <summary>PDT-01</summary>
	{attribute 'OPC.UA.DA' := '1'}  				                
	filter_diff_pres_min												: REAL;
    /// <summary>PDT-01</summary>
	{attribute 'OPC.UA.DA' := '1'}  				                
	filter_diff_pres_offset												: REAL;

    /// <summary>PDT-02</summary>
	{attribute 'OPC.UA.DA' := '1'}  				                
	sorbent_diff_pres_low												: REAL;
    /// <summary>PDT-02</summary>
	{attribute 'OPC.UA.DA' := '1'}  				                
	sorbent_diff_pres_high												: REAL;
    /// <summary>PDT-02</summary>
	{attribute 'OPC.UA.DA' := '1'}  				                
	sorbent_diff_pres_min												: REAL;
    /// <summary>PDT-02</summary>
	{attribute 'OPC.UA.DA' := '1'}  				                
	sorbent_diff_pres_offset											: REAL;

    /// <summary>PDT-03</summary>
	{attribute 'OPC.UA.DA' := '1'}  				                
	fan_diff_pres_low													: REAL;
    /// <summary>PDT-03</summary>
	{attribute 'OPC.UA.DA' := '1'}  				                
	fan_diff_pres_high													: REAL;
    /// <summary>PDT-03</summary>
	{attribute 'OPC.UA.DA' := '1'}  				                
	fan_diff_pres_min													: REAL;
    /// <summary>PDT-03</summary>
	{attribute 'OPC.UA.DA' := '1'}  				                
	fan_diff_pres_offset												: REAL;

    /// <summary>PT-01</summary>
	{attribute 'OPC.UA.DA' := '1'}  				                
	reactor_pres_low													: REAL;
    /// <summary>PT-01</summary>
	{attribute 'OPC.UA.DA' := '1'}  				                
	reactor_pres_high													: REAL;
    /// <summary>PT-01</summary>
	{attribute 'OPC.UA.DA' := '1'}  				                
	reactor_pres_min													: REAL;
    /// <summary>PT-01</summary>
	{attribute 'OPC.UA.DA' := '1'}  				                
	reactor_pres_offset													: REAL;

    /// <summary>TT04</summary>
	{attribute 'OPC.UA.DA' := '1'}  				                
	air_inlet_temp_offset												: REAL;

    /// <summary>TT05</summary>
	{attribute 'OPC.UA.DA' := '1'}  				                
	reactor_wall_temp_offset											: REAL;

    /// <summary>01-TT-01</summary>
	{attribute 'OPC.UA.DA' := '1'}  				                
	cart01_front_temp_offset											: REAL;
    /// <summary>10-TT-03</summary>
	{attribute 'OPC.UA.DA' := '1'}  				                
	cart01_back_temp_offset												: REAL;
    /// <summary>02-TT-01</summary>
	{attribute 'OPC.UA.DA' := '1'}  				                
	cart02_front_temp_offset											: REAL;
    /// <summary>02-TT-03</summary>
	{attribute 'OPC.UA.DA' := '1'}  				                
	cart02_back_temp_offset												: REAL;
    /// <summary>03-TT-01</summary>
	{attribute 'OPC.UA.DA' := '1'}  				                
	cart03_front_temp_offset											: REAL;
    /// <summary>03-TT-03</summary>
	{attribute 'OPC.UA.DA' := '1'}  				                
	cart03_back_temp_offset												: REAL;
    /// <summary>04-TT-01</summary>
	{attribute 'OPC.UA.DA' := '1'}  				                
	cart04_front_temp_offset											: REAL;
    /// <summary>04-TT-03</summary>
	{attribute 'OPC.UA.DA' := '1'}  				                
	cart04_back_temp_offset												: REAL;
    /// <summary>05-TT-01</summary>
	{attribute 'OPC.UA.DA' := '1'}  				                
	cart05_front_temp_offset											: REAL;
    /// <summary>05-TT-03</summary>
	{attribute 'OPC.UA.DA' := '1'}  				                
	cart05_back_temp_offset												: REAL;
    /// <summary>06-TT-01</summary>
	{attribute 'OPC.UA.DA' := '1'}  				                
	cart06_front_temp_offset											: REAL;
    /// <summary>06-TT-03</summary>
	{attribute 'OPC.UA.DA' := '1'}  				                
	cart06_back_temp_offset												: REAL;
    /// <summary>07-TT-01</summary>
	{attribute 'OPC.UA.DA' := '1'}  				                
	cart07_front_temp_offset											: REAL;
    /// <summary>07-TT-03</summary>
	{attribute 'OPC.UA.DA' := '1'}  				                
	cart07_back_temp_offset												: REAL;
    /// <summary>08-TT-01</summary>
	{attribute 'OPC.UA.DA' := '1'}  				                
	cart08_front_temp_offset											: REAL;
    /// <summary>08-TT-03</summary>
	{attribute 'OPC.UA.DA' := '1'}  				                
	cart08_back_temp_offset												: REAL;
    /// <summary>09-TT-01</summary>
	{attribute 'OPC.UA.DA' := '1'}  				                
	cart09_front_temp_offset											: REAL;
    /// <summary>09-TT-03</summary>
	{attribute 'OPC.UA.DA' := '1'}  				                
	cart09_back_temp_offset												: REAL;
    /// <summary>10-TT-01</summary>
	{attribute 'OPC.UA.DA' := '1'}  				                
	cart10_front_temp_offset											: REAL;
    /// <summary>10-TT-03</summary>
	{attribute 'OPC.UA.DA' := '1'}  				                
	cart10_back_temp_offset												: REAL;
    /// <summary>11-TT-01</summary>
	{attribute 'OPC.UA.DA' := '1'}  				                
	cart11_front_temp_offset											: REAL;
    /// <summary>11-TT-03</summary>
	{attribute 'OPC.UA.DA' := '1'}  				                
	cart11_back_temp_offset												: REAL;
    /// <summary>12-TT-01</summary>
	{attribute 'OPC.UA.DA' := '1'}  				                
	cart12_front_temp_offset											: REAL;
    /// <summary>12-TT-03</summary>
	{attribute 'OPC.UA.DA' := '1'}  				                
	cart12_back_temp_offset												: REAL;
	
END_VAR

// Theseus - FB_Reactor
// Rev 1.0 - November 4, 2024

inlet_co2																:= F_AnalogIn(AT_01, inlet_co2_low, inlet_co2_high, inlet_co2_min, inlet_co2_offset);
inlet_co2_error															:= AT_01_error AND NOT _InletCO2ErrorOff;

inlet_h2o																:= F_AnalogIn(AT_02, inlet_h2o_low, inlet_h2o_high, inlet_h2o_min, inlet_h2o_offset);
inlet_h2o_error															:= AT_02_error AND NOT _InletH2OErrorOff;

outlet_co2																:= F_AnalogIn(AT_03, outlet_co2_low, outlet_co2_high, outlet_co2_min, outlet_co2_offset);
outlet_co2_error														:= AT_03_error AND NOT _OutletCO2ErrorOff;

outlet_h2o																:= F_AnalogIn(AT_04, outlet_h2o_low, outlet_h2o_high, outlet_h2o_min, outlet_h2o_offset);
outlet_h2o_error														:= AT_04_error AND NOT _OutletH2OErrorOff;

reactor_pres															:= F_AnalogIn(PT_01, reactor_pres_low, reactor_pres_high, reactor_pres_min, reactor_pres_offset);
reactor_pres_error														:= PT_01_error AND NOT _ReactorPresErrorOff;

air_flow																:= F_AnalogIn(FT_01, air_flow_low, air_flow_high, air_flow_min, air_flow_offset);
air_flow_error															:= FT_01_error AND NOT _AirFlowErrorOff;

filter_diff_pres														:= F_AnalogIn(PDT_01, filter_diff_pres_low, filter_diff_pres_high, filter_diff_pres_min, filter_diff_pres_offset);
filter_diff_pres_error													:= PDT_01_error AND NOT _FilterDiffPresErrorOff;

sorbent_diff_pres														:= F_AnalogIn(PDT_02, sorbent_diff_pres_low, sorbent_diff_pres_high, sorbent_diff_pres_min, sorbent_diff_pres_offset);
sorbent_diff_pres_error													:= PDT_02_error AND NOT _SorbentDiffPresErrorOff;

fan_diff_pres															:= F_AnalogIn(PDT_03, fan_diff_pres_low, fan_diff_pres_high, fan_diff_pres_min, fan_diff_pres_offset);
fan_diff_pres_error														:= PDT_03_error AND NOT _FanDiffPresErrorOff;

air_inlet_temp															:= F_Temperature(TT_04, air_inlet_temp_offset);
air_inlet_temp_error													:= TT_04_error AND NOT _AirInletTempErrorOff;

reactor_wall_temp														:= F_Temperature(TT_05, reactor_wall_temp_offset);
reactor_wall_temp_error													:= TT_05_error AND NOT _ReactorWallTempErrorOff;

AT_01_pump																:= inlet_co2_pump;
inlet_co2_pump_cmd_status												:= AT_01_pump;

AT_01_sol																:= inlet_co2_sol;
inlet_co2_sol_cmd_status												:= AT_01_sol;

AT_03_pump																:= outlet_co2_pump;
outlet_co2_pump_cmd_status												:= AT_03_pump;
                                                                           
AT_03_sol																:= outlet_co2_sol;
outlet_co2_sol_cmd_status												:= AT_03_sol;

// SORBENT TEMPERATURE HANDLING
rtrigSorbentErrorCheck(CLK:= MAIN.bHalfSecondPulse);
IF rtrigSorbentErrorCheck.Q THEN
	A_Sorbent_Temperatures();
END_IF

XV_02																	:= repres_valve;
repres_valve_open_cmd_status											:= XV_02;
repres_valve_clear														:= F_ValveClear(repres_valve, repres_valve_open, repres_valve_closed);

XV_09																	:= over_pressure_test_control;
over_pressure_test_control_cmd_status									:= XV_09;

// FAN
tonFan(IN:= fan_vfd_setpoint <> rFanSPOld, PT:= INT_TO_TIME((unit - 1) * _FAN_DELAY_TIME));
IF tonFan.Q THEN
	rfanSPOld															:= fan_vfd_setpoint;
	rRpm																:= fan_vfd_setpoint * _FAN_RPM_FACTOR;
END_IF
fb_Fan(	Enable_Vfd														:= NOT fan_vfd_ecat_state AND fan_vfd_enable,
		Fault_Reset														:= fan_vfd_reset, 
		Rpm																:= rRpm, 
		Minimum_Speed													:= _FAN_SPEED_MIN,
		Maximum_Speed													:= _FAN_SPEED_MAX, 
		StatusWord														:= fan_vfd_status, 
		ControlWord														=> fan_vfd_control, 
		TargetRpm														=> fan_vfd_target_vel, 
		Ready															=> fan_vfd_enabled,
		Error															=> fan_vfd_error);
fan_vfd_output															:= WORD_TO_REAL(fan_vfd_velocity) / _FAN_RPM_FACTOR;
fan_vfd_output_current													:= DINT_TO_REAL(fan_vfd_current)/100;
IF fan_vfd_reset THEN
	fan_vfd_reset														:= FALSE;
END_IF

// CLAMPS & DOORS
fbInletDoorsClosed(valve:= inlet_door_close_valve, limit_switch:= inlet_door_near_closed_ls AND inlet_door_far_closed_ls, door_closed=> inlet_doors_closed);
fbOutletDoorsClosed(valve:= outlet_door_close_valve, limit_switch:= outlet_door_near_closed_ls AND outlet_door_far_closed_ls, door_closed=> outlet_doors_closed);

inlet_doors_open														:= inlet_door_near_open_ls AND inlet_door_far_open_ls;
outlet_doors_open														:= outlet_door_near_open_ls AND outlet_door_far_open_ls;

inlet_door_clamps_extended												:= inlet_door_near_clamps_extended AND inlet_door_far_clamps_extended;
inlet_door_clamps_retracted												:= NOT inlet_door_near_clamps_extended AND NOT inlet_door_far_clamps_extended;
outlet_door_clamps_extended												:= outlet_door_near_clamps_extended AND outlet_door_far_clamps_extended;
outlet_door_clamps_retracted											:= NOT outlet_door_near_clamps_extended AND NOT outlet_door_far_clamps_extended;
 
IF extend_inlet_door_clamps THEN
	inlet_door_near_clamps_retract_valve								:= FALSE;
	inlet_door_far_clamps_retract_valve									:= FALSE;
	inlet_door_near_clamps_extend_valve									:= TRUE;
	inlet_door_far_clamps_extend_valve									:= TRUE;
ELSIF retract_inlet_door_clamps THEN
	inlet_door_near_clamps_extend_valve									:= FALSE;
	inlet_door_far_clamps_extend_valve									:= FALSE;
	inlet_door_near_clamps_retract_valve								:= TRUE;
	inlet_door_far_clamps_retract_valve									:= TRUE;
END_IF
IF extend_outlet_door_clamps THEN
	outlet_door_near_clamps_retract_valve								:= FALSE;
	outlet_door_far_clamps_retract_valve								:= FALSE;
	outlet_door_near_clamps_extend_valve								:= TRUE;
	outlet_door_far_clamps_extend_valve									:= TRUE;
ELSIF retract_outlet_door_clamps THEN
	outlet_door_near_clamps_extend_valve								:= FALSE;
	outlet_door_far_clamps_extend_valve									:= FALSE;
	outlet_door_near_clamps_retract_valve								:= TRUE;
	outlet_door_far_clamps_retract_valve								:= TRUE;
END_IF

extend_inlet_door_clamps												:= FALSE;
retract_inlet_door_clamps												:= FALSE;
extend_outlet_door_clamps												:= FALSE;
retract_outlet_door_clamps												:= FALSE;

IF open_inlet_door THEN
	inlet_door_open_valve												:= TRUE;
	inlet_door_close_valve												:= FALSE;
ELSIF close_inlet_door THEN
	inlet_door_close_valve												:= TRUE;
	inlet_door_open_valve												:= FALSE;
END_IF
IF open_outlet_door THEN
	outlet_door_open_valve												:= TRUE;
	outlet_door_close_valve												:= FALSE;
ELSIF close_outlet_door THEN
	outlet_door_close_valve												:= TRUE;
	outlet_door_open_valve												:= FALSE;
END_IF

open_inlet_door															:= FALSE;
close_inlet_door														:= FALSE;
open_outlet_door														:= FALSE;
close_outlet_door														:= FALSE;

temp_low																:=sorbent_low_temp		;   
temp_high       														:=sorbent_high_temp		; 
temp_average    														:=sorbent_average_temp	;

ACTION A_Sorbent_Temperatures:
// Theseus - FB_ReatorIO.A_Sorbent_Temperatures
// Rev 1.0 - October 8, 2024

sorbent_low_temp														:= 1000;
sorbent_high_temp														:= -1000;

rTempTotal																:= 0;
iTempCount																:= 0;

cart01_front_temp														:= F_Temperature(_01_TT_01, cart01_front_temp_offset);
cart01_front_temp_error 												:= _01_TT_01_error OR iCount[0] < 30;
cart01_back_temp														:= F_Temperature(_01_TT_03, cart01_back_temp_offset);
cart01_back_temp_error 													:= _01_TT_03_Error OR iCount[1] < 30;
cart01_temp_front_calc(Error:= cart01_front_temp_error, Temp:= cart01_front_temp, Low:= sorbent_low_temp, High:= sorbent_high_temp, Total:= rTempTotal, Counter:= iTempCount);
cart01_temp_back_calc(Error:= cart01_back_temp_error, Temp:= cart01_back_temp, Low:= sorbent_low_temp, High:= sorbent_high_temp, Total:= rTempTotal, Counter:= iTempCount);

cart02_front_temp														:= F_Temperature(_02_TT_01, cart02_front_temp_offset);
cart02_front_temp_error 												:= _02_TT_01_error OR iCount[2] < 30;
cart02_back_temp														:= F_Temperature(_02_TT_03, cart02_back_temp_offset);
cart02_back_temp_error 													:= _02_TT_03_Error OR iCount[3] < 30;
cart02_temp_front_calc(Error:= cart02_front_temp_error, Temp:= cart02_front_temp, Low:= sorbent_low_temp, High:= sorbent_high_temp, Total:= rTempTotal, Counter:= iTempCount);
cart02_temp_back_calc(Error:= cart02_back_temp_error, Temp:= cart02_back_temp, Low:= sorbent_low_temp, High:= sorbent_high_temp, Total:= rTempTotal, Counter:= iTempCount);

cart03_front_temp														:= F_Temperature(_03_TT_01, cart03_front_temp_offset);
cart03_front_temp_error 												:= _03_TT_01_error OR iCount[4] < 30;
cart03_back_temp														:= F_Temperature(_03_TT_03, cart03_back_temp_offset);
cart03_back_temp_error 													:= _03_TT_03_Error OR iCount[5] < 30;
cart03_temp_front_calc(Error:= cart03_front_temp_error, Temp:= cart03_front_temp, Low:= sorbent_low_temp, High:= sorbent_high_temp, Total:= rTempTotal, Counter:= iTempCount);
cart03_temp_back_calc(Error:= cart03_back_temp_error, Temp:= cart03_back_temp, Low:= sorbent_low_temp, High:= sorbent_high_temp, Total:= rTempTotal, Counter:= iTempCount);

cart04_front_temp														:= F_Temperature(_04_TT_01, cart04_front_temp_offset);
cart04_front_temp_error 												:= _04_TT_01_error OR iCount[6] < 30;
cart04_back_temp														:= F_Temperature(_04_TT_03, cart04_back_temp_offset);
cart04_back_temp_error 													:= _04_TT_03_Error OR iCount[7] < 30;
cart04_temp_front_calc(Error:= cart04_front_temp_error, Temp:= cart04_front_temp, Low:= sorbent_low_temp, High:= sorbent_high_temp, Total:= rTempTotal, Counter:= iTempCount);
cart04_temp_back_calc(Error:= cart04_back_temp_error, Temp:= cart04_back_temp, Low:= sorbent_low_temp, High:= sorbent_high_temp, Total:= rTempTotal, Counter:= iTempCount);

cart05_front_temp														:= F_Temperature(_05_TT_01, cart05_front_temp_offset);
cart05_front_temp_error 												:= _05_TT_01_error OR iCount[8] < 30;
cart05_back_temp														:= F_Temperature(_05_TT_03, cart05_back_temp_offset);
cart05_back_temp_error 													:= _05_TT_03_Error OR iCount[9] < 30;
cart05_temp_front_calc(Error:= cart05_front_temp_error, Temp:= cart05_front_temp, Low:= sorbent_low_temp, High:= sorbent_high_temp, Total:= rTempTotal, Counter:= iTempCount);
cart05_temp_back_calc(Error:= cart05_back_temp_error, Temp:= cart05_back_temp, Low:= sorbent_low_temp, High:= sorbent_high_temp, Total:= rTempTotal, Counter:= iTempCount);

cart06_front_temp														:= F_Temperature(_06_TT_01, cart06_front_temp_offset);
cart06_front_temp_error 												:= _06_TT_01_error OR iCount[10] < 30;
cart06_back_temp														:= F_Temperature(_06_TT_03, cart06_back_temp_offset);
cart06_back_temp_error 													:= _06_TT_03_Error OR iCount[11] < 30;
cart06_temp_front_calc(Error:= cart06_front_temp_error, Temp:= cart06_front_temp, Low:= sorbent_low_temp, High:= sorbent_high_temp, Total:= rTempTotal, Counter:= iTempCount);
cart06_temp_back_calc(Error:= cart06_back_temp_error, Temp:= cart06_back_temp, Low:= sorbent_low_temp, High:= sorbent_high_temp, Total:= rTempTotal, Counter:= iTempCount);

cart07_front_temp														:= F_Temperature(_07_TT_01, cart07_front_temp_offset);
cart07_front_temp_error 												:= _07_TT_01_error OR iCount[12] < 30;
cart07_back_temp														:= F_Temperature(_07_TT_03, cart07_back_temp_offset);
cart07_back_temp_error 													:= _07_TT_03_Error OR iCount[13] < 30;
cart07_temp_front_calc(Error:= cart07_front_temp_error, Temp:= cart07_front_temp, Low:= sorbent_low_temp, High:= sorbent_high_temp, Total:= rTempTotal, Counter:= iTempCount);
cart07_temp_back_calc(Error:= cart07_back_temp_error, Temp:= cart07_back_temp, Low:= sorbent_low_temp, High:= sorbent_high_temp, Total:= rTempTotal, Counter:= iTempCount);

cart08_front_temp														:= F_Temperature(_08_TT_01, cart08_front_temp_offset);
cart08_front_temp_error 												:= _08_TT_01_error OR iCount[14] < 30;
cart08_back_temp														:= F_Temperature(_08_TT_03, cart08_back_temp_offset);
cart08_back_temp_error 													:= _08_TT_03_Error OR iCount[15] < 30;
cart08_temp_front_calc(Error:= cart08_front_temp_error, Temp:= cart08_front_temp, Low:= sorbent_low_temp, High:= sorbent_high_temp, Total:= rTempTotal, Counter:= iTempCount);
cart08_temp_back_calc(Error:= cart08_back_temp_error, Temp:= cart08_back_temp, Low:= sorbent_low_temp, High:= sorbent_high_temp, Total:= rTempTotal, Counter:= iTempCount);

cart09_front_temp														:= F_Temperature(_09_TT_01, cart09_front_temp_offset);
cart09_front_temp_error 												:= _09_TT_01_error OR iCount[16] < 30;
cart09_back_temp														:= F_Temperature(_09_TT_03, cart09_back_temp_offset);
cart09_back_temp_error 													:= _09_TT_03_Error OR iCount[17] < 30;
cart09_temp_front_calc(Error:= cart09_front_temp_error, Temp:= cart09_front_temp, Low:= sorbent_low_temp, High:= sorbent_high_temp, Total:= rTempTotal, Counter:= iTempCount);
cart09_temp_back_calc(Error:= cart09_back_temp_error, Temp:= cart09_back_temp, Low:= sorbent_low_temp, High:= sorbent_high_temp, Total:= rTempTotal, Counter:= iTempCount);

